LIN {X 0,Y 466.685,Z 325.228,A -85,B 0,C 180,E1 -7652.59,E2 -7652.59} C_VEL
LIN {X 0,Y 466.715,Z 322.29,A -85,B 0,C 180,E1 -7653.886,E2 -7653.886} C_VEL
LIN {X 0,Y 466.717,Z 319.594,A -85,B 0,C 180,E1 -7654.751,E2 -7654.751} C_VEL
LIN {X 0,Y 466.821,Z 316.273,A -85,B 0,C 180,E1 -7655.616,E2 -7655.616} C_VEL
LIN {X 0,Y 466.891,Z 311.9,A -85,B 0,C 180,E1 -7656.544,E2 -7656.544} C_VEL
LIN {X 0,Y 467.057,Z 305.94,A -85,B 0,C 180,E1 -7657.566,E2 -7657.566} C_VEL
LIN {X 0,Y 467.255,Z 299.775,A -85,B 0,C 180,E1 -7658.433,E2 -7658.433} C_VEL
LIN {X 0,Y 467.469,Z 293.294,A -85,B 0,C 180,E1 -7659.192,E2 -7659.192} C_VEL
LIN {X 0,Y 467.75,Z 285.446,A -85,B 0,C 180,E1 -7659.95,E2 -7659.95} C_VEL
LIN {X 0,Y 468.086,Z 277.17,A -85,B 0,C 180,E1 -7660.599,E2 -7660.599} C_VEL
LIN {X 0,Y 468.393,Z 266.639,A -85,B 0,C 180,E1 -7661.248,E2 -7661.248} C_VEL
LIN {X 0,Y 468.216,Z 258.863,A -85,B 0,C 180,E1 -7661.613,E2 -7661.613} C_VEL
LIN {X 0,Y 466.947,Z 246.747,A -85,B 0,C 180,E1 -7662.034,E2 -7662.034} C_VEL
LIN {X 0,Y 466.898,Z 245.995,A -85,B 0,C 180,E1 -7662.074,E2 -7662.074} C_VEL
LIN {X 0,Y 467.105,Z 234.959,A -85,B 0,C 180,E1 -7665.714,E2 -7665.714} C_VEL
LIN {X 0,Y 467.312,Z 226.159,A -85,B 0,C 180,E1 -7668.653,E2 -7668.653} C_VEL
LIN {X 0,Y 467.611,Z 217.438,A -85,B 0,C 180,E1 -7671.619,E2 -7671.619} C_VEL
LIN {X 0,Y 468.104,Z 206.857,A -85,B 0,C 180,E1 -7675.304,E2 -7675.304} C_VEL
LIN {X 0,Y 468.59,Z 197.452,A -85,B 0,C 180,E1 -7678.682,E2 -7678.682} C_VEL
LIN {X 0,Y 468.856,Z 190.408,A -85,B 0,C 180,E1 -7681.305,E2 -7681.305} C_VEL
LIN {X 0,Y 467.631,Z 183.051,A -85,B 0,C 180,E1 -7684.249,E2 -7684.249} C_VEL
LIN {X 0,Y 467.551,Z 183.059,A -85,B 0,C 180,E1 -7687.186,E2 -7687.186} C_VEL
LIN {X 0,Y 467.578,Z 183.056,A -85,B 0,C 180,E1 -7690.265,E2 -7690.265} C_VEL
LIN {X 0,Y 467.59,Z 183.054,A -85,B 0,C 180,E1 -7692.567,E2 -7692.567} C_VEL
LIN {X 0,Y 467.569,Z 183.056,A -85,B 0,C 180,E1 -7695.052,E2 -7695.052} C_VEL
LIN {X 0,Y 467.577,Z 183.055,A -85,B 0,C 180,E1 -7698.597,E2 -7698.597} C_VEL
LIN {X 0,Y 467.569,Z 183.058,A -85,B 0,C 180,E1 -7701.955,E2 -7701.955} C_VEL
LIN {X 0,Y 467.568,Z 183.054,A -85,B 0,C 180,E1 -7705.167,E2 -7705.167} C_VEL
LIN {X 0,Y 467.587,Z 183.056,A -85,B 0,C 180,E1 -7708.26,E2 -7708.26} C_VEL
LIN {X 0,Y 467.579,Z 183.055,A -85,B 0,C 180,E1 -7711.25,E2 -7711.25} C_VEL
LIN {X 0,Y 467.602,Z 183.053,A -85,B 0,C 180,E1 -7714.159,E2 -7714.159} C_VEL
LIN {X 0,Y 467.581,Z 183.054,A -85,B 0,C 180,E1 -7716.996,E2 -7716.996} C_VEL
LIN {X 0,Y 467.627,Z 183.051,A -85,B 0,C 180,E1 -7719.777,E2 -7719.777} C_VEL
LIN {X 0,Y 467.603,Z 183.051,A -85,B 0,C 180,E1 -7722.506,E2 -7722.506} C_VEL
LIN {X 0,Y 467.611,Z 183.052,A -85,B 0,C 180,E1 -7725.196,E2 -7725.196} C_VEL
LIN {X 0,Y 467.661,Z 183.045,A -85,B 0,C 180,E1 -7727.854,E2 -7727.854} C_VEL
LIN {X 0,Y 467.673,Z 183.045,A -85,B 0,C 180,E1 -7731.356,E2 -7731.356} C_VEL
LIN {X 0,Y 467.736,Z 183.035,A -85,B 0,C 180,E1 -7733.962,E2 -7733.962} C_VEL
LIN {X 0,Y 467.861,Z 183.022,A -85,B 0,C 180,E1 -7737.416,E2 -7737.416} C_VEL
LIN {X 0,Y 467.885,Z 183.017,A -85,B 0,C 180,E1 -7739.999,E2 -7739.999} C_VEL
LIN {X 0,Y 467.861,Z 183.019,A -85,B 0,C 180,E1 -7742.582,E2 -7742.582} C_VEL
LIN {X 0,Y 467.736,Z 183.033,A -85,B 0,C 180,E1 -7746.037,E2 -7746.037} C_VEL
LIN {X 0,Y 467.672,Z 183.043,A -85,B 0,C 180,E1 -7748.642,E2 -7748.642} C_VEL
LIN {X 0,Y 467.658,Z 183.045,A -85,B 0,C 180,E1 -7752.144,E2 -7752.144} C_VEL
LIN {X 0,Y 467.64,Z 183.047,A -85,B 0,C 180,E1 -7755.694,E2 -7755.694} C_VEL
LIN {X 0,Y 467.623,Z 183.05,A -85,B 0,C 180,E1 -7759.307,E2 -7759.307} C_VEL
LIN {X 0,Y 467.535,Z 183.062,A -85,B 0,C 180,E1 -7762.073,E2 -7762.073} C_VEL
LIN {X 0,Y 467.585,Z 183.054,A -85,B 0,C 180,E1 -7764.887,E2 -7764.887} C_VEL
LIN {X 0,Y 467.627,Z 183.048,A -85,B 0,C 180,E1 -7767.767,E2 -7767.767} C_VEL
LIN {X 0,Y 467.567,Z 183.056,A -85,B 0,C 180,E1 -7771.044,E2 -7771.044} C_VEL
LIN {X 0,Y 467.588,Z 183.054,A -85,B 0,C 180,E1 -7774.241,E2 -7774.241} C_VEL
LIN {X 0,Y 467.547,Z 183.059,A -85,B 0,C 180,E1 -7777.186,E2 -7777.186} C_VEL
LIN {X 0,Y 467.574,Z 183.056,A -85,B 0,C 180,E1 -7780.264,E2 -7780.264} C_VEL
LIN {X 0,Y 467.582,Z 183.054,A -85,B 0,C 180,E1 -7782.566,E2 -7782.566} C_VEL
LIN {X 0,Y 467.566,Z 183.056,A -85,B 0,C 180,E1 -7785.052,E2 -7785.052} C_VEL
LIN {X 0,Y 467.584,Z 183.055,A -85,B 0,C 180,E1 -7787.439,E2 -7787.439} C_VEL
LIN {X 0,Y 467.576,Z 183.054,A -85,B 0,C 180,E1 -7790.854,E2 -7790.854} C_VEL
LIN {X 0,Y 467.557,Z 183.057,A -85,B 0,C 180,E1 -7794.259,E2 -7794.259} C_VEL
LIN {X 0,Y 467.576,Z 183.055,A -85,B 0,C 180,E1 -7797.32,E2 -7797.32} C_VEL
LIN {X 0,Y 467.572,Z 183.055,A -85,B 0,C 180,E1 -7800.665,E2 -7800.665} C_VEL
LIN {X 0,Y 467.609,Z 183.052,A -85,B 0,C 180,E1 -7803.199,E2 -7803.199} C_VEL
LIN {X 0,Y 467.585,Z 183.054,A -85,B 0,C 180,E1 -7806.467,E2 -7806.467} C_VEL
LIN {X 0,Y 467.616,Z 183.05,A -85,B 0,C 180,E1 -7809.777,E2 -7809.777} C_VEL
LIN {X 0,Y 467.601,Z 183.051,A -85,B 0,C 180,E1 -7812.506,E2 -7812.506} C_VEL
LIN {X 0,Y 467.594,Z 183.052,A -85,B 0,C 180,E1 -7815.417,E2 -7815.417} C_VEL
LIN {X 0,Y 466.928,Z 183.134,A -85,B 0,C 180,E1 -7816.137,E2 -7816.137} C_VEL
LIN {X 0,Y 464.094,Z 183.489,A -85,B 0,C 180,E1 -7817.306,E2 -7817.306} C_VEL
LIN {X 0,Y 461.696,Z 183.788,A -85,B 0,C 180,E1 -7818.248,E2 -7818.248} C_VEL
LIN {X 0,Y 460.666,Z 183.917,A -85,B 0,C 180,E1 -7818.976,E2 -7818.976} C_VEL
LIN {X 0,Y 460.581,Z 183.926,A -85,B 0,C 180,E1 -7819.223,E2 -7819.223} C_VEL
LIN {X 0,Y 460.711,Z 183.91,A -85,B 0,C 180,E1 -7822.538,E2 -7822.538} C_VEL
LIN {X 0,Y 460.689,Z 183.915,A -85,B 0,C 180,E1 -7824.748,E2 -7824.748} C_VEL
LIN {X 0,Y 460.79,Z 183.9,A -85,B 0,C 180,E1 -7827.377,E2 -7827.377} C_VEL
LIN {X 0,Y 460.842,Z 183.894,A -85,B 0,C 180,E1 -7830,E2 -7830} C_VEL
LIN {X 0,Y 460.817,Z 183.898,A -85,B 0,C 180,E1 -7832.622,E2 -7832.622} C_VEL
LIN {X 0,Y 460.702,Z 183.913,A -85,B 0,C 180,E1 -7836.13,E2 -7836.13} C_VEL
LIN {X 0,Y 460.62,Z 183.922,A -85,B 0,C 180,E1 -7838.776,E2 -7838.776} C_VEL
LIN {X 0,Y 460.59,Z 183.928,A -85,B 0,C 180,E1 -7842.335,E2 -7842.335} C_VEL
LIN {X 0,Y 460.291,Z 184.096,A -85,B 0,C 180,E1 -7844.931,E2 -7844.931} C_VEL
LIN {X 0,Y 460.115,Z 188.342,A -85,B 0,C 180,E1 -7847.787,E2 -7847.787} C_VEL
LIN {X 0,Y 460.039,Z 192.537,A -85,B 0,C 180,E1 -7850.571,E2 -7850.571} C_VEL
LIN {X 0,Y 459.941,Z 197.069,A -85,B 0,C 180,E1 -7853.539,E2 -7853.539} C_VEL
LIN {X 0,Y 459.84,Z 201.353,A -85,B 0,C 180,E1 -7856.31,E2 -7856.31} C_VEL
LIN {X 0,Y 459.729,Z 206.164,A -85,B 0,C 180,E1 -7859.384,E2 -7859.384} C_VEL
LIN {X 0,Y 459.676,Z 211.565,A -85,B 0,C 180,E1 -7862.767,E2 -7862.767} C_VEL
LIN {X 0,Y 459.686,Z 213.246,A -85,B 0,C 180,E1 -7863.722,E2 -7863.722} C_VEL
LIN {X 0,Y 461.221,Z 222.711,A -85,B 0,C 180,E1 -7864.121,E2 -7864.121} C_VEL
LIN {X 0,Y 461.594,Z 228.119,A -85,B 0,C 180,E1 -7864.388,E2 -7864.388} C_VEL
LIN {X 0,Y 461.262,Z 237.826,A -85,B 0,C 180,E1 -7864.994,E2 -7864.994} C_VEL
LIN {X 0,Y 461.001,Z 245.945,A -85,B 0,C 180,E1 -7865.644,E2 -7865.644} C_VEL
LIN {X 0,Y 460.712,Z 254.566,A -85,B 0,C 180,E1 -7866.508,E2 -7866.508} C_VEL
LIN {X 0,Y 460.38,Z 262.083,A -85,B 0,C 180,E1 -7867.459,E2 -7867.459} C_VEL
LIN {X 0,Y 460.171,Z 268.447,A -85,B 0,C 180,E1 -7868.488,E2 -7868.488} C_VEL
LIN {X 0,Y 459.974,Z 272.818,A -85,B 0,C 180,E1 -7869.351,E2 -7869.351} C_VEL
LIN {X 0,Y 459.837,Z 276.248,A -85,B 0,C 180,E1 -7870.167,E2 -7870.167} C_VEL
LIN {X 0,Y 459.689,Z 280.407,A -85,B 0,C 180,E1 -7871.486,E2 -7871.486} C_VEL
LIN {X 0,Y 459.591,Z 283.196,A -85,B 0,C 180,E1 -7872.778,E2 -7872.778} C_VEL
LIN {X 0,Y 459.544,Z 284.733,A -85,B 0,C 180,E1 -7874.047,E2 -7874.047} C_VEL
LIN {X 0,Y 459.523,Z 285.066,A -85,B 0,C 180,E1 -7875.291,E2 -7875.291} C_VEL
LIN {X 0,Y 459.57,Z 284.346,A -85,B 0,C 180,E1 -7876.517,E2 -7876.517} C_VEL
LIN {X 0,Y 459.622,Z 282.626,A -85,B 0,C 180,E1 -7877.718,E2 -7877.718} C_VEL
LIN {X 0,Y 459.713,Z 279.899,A -85,B 0,C 180,E1 -7878.902,E2 -7878.902} C_VEL
LIN {X 0,Y 459.936,Z 274.892,A -85,B 0,C 180,E1 -7880.362,E2 -7880.362} C_VEL
LIN {X 0,Y 460.183,Z 269.452,A -85,B 0,C 180,E1 -7881.514,E2 -7881.514} C_VEL
LIN {X 0,Y 460.417,Z 263.346,A -85,B 0,C 180,E1 -7882.537,E2 -7882.537} C_VEL
LIN {X 0,Y 460.766,Z 255.068,A -85,B 0,C 180,E1 -7883.622,E2 -7883.622} C_VEL
LIN {X 0,Y 461.056,Z 246.575,A -85,B 0,C 180,E1 -7884.484,E2 -7884.484} C_VEL
LIN {X 0,Y 461.339,Z 238.745,A -85,B 0,C 180,E1 -7885.121,E2 -7885.121} C_VEL
LIN {X 0,Y 461.681,Z 229.369,A -85,B 0,C 180,E1 -7885.721,E2 -7885.721} C_VEL
LIN {X 0,Y 461.438,Z 223.284,A -85,B 0,C 180,E1 -7886.03,E2 -7886.03} C_VEL
LIN {X 0,Y 459.731,Z 213.544,A -85,B 0,C 180,E1 -7886.48,E2 -7886.48} C_VEL
LIN {X 0,Y 459.77,Z 208.543,A -85,B 0,C 180,E1 -7889.707,E2 -7889.707} C_VEL
LIN {X 0,Y 459.922,Z 203.907,A -85,B 0,C 180,E1 -7892.716,E2 -7892.716} C_VEL
LIN {X 0,Y 460,Z 199.515,A -85,B 0,C 180,E1 -7895.638,E2 -7895.638} C_VEL
LIN {X 0,Y 460.104,Z 194.897,A -85,B 0,C 180,E1 -7898.711,E2 -7898.711} C_VEL
LIN {X 0,Y 460.227,Z 191.101,A -85,B 0,C 180,E1 -7901.297,E2 -7901.297} C_VEL
LIN {X 0,Y 460.332,Z 186.977,A -85,B 0,C 180,E1 -7904.12,E2 -7904.12} C_VEL
LIN {X 0,Y 460.347,Z 184.5,A -85,B 0,C 180,E1 -7905.862,E2 -7905.862} C_VEL
LIN {X 0,Y 460.432,Z 183.952,A -85,B 0,C 180,E1 -7906.765,E2 -7906.765} C_VEL
LIN {X 0,Y 460.603,Z 183.928,A -85,B 0,C 180,E1 -7908.56,E2 -7908.56} C_VEL
LIN {X 0,Y 460.696,Z 183.917,A -85,B 0,C 180,E1 -7912.109,E2 -7912.109} C_VEL
LIN {X 0,Y 460.697,Z 183.917,A -85,B 0,C 180,E1 -7914.749,E2 -7914.749} C_VEL
LIN {X 0,Y 460.801,Z 183.901,A -85,B 0,C 180,E1 -7917.378,E2 -7917.378} C_VEL
LIN {X 0,Y 460.855,Z 183.894,A -85,B 0,C 180,E1 -7920.001,E2 -7920.001} C_VEL
LIN {X 0,Y 460.801,Z 183.9,A -85,B 0,C 180,E1 -7922.623,E2 -7922.623} C_VEL
LIN {X 0,Y 460.709,Z 183.912,A -85,B 0,C 180,E1 -7926.131,E2 -7926.131} C_VEL
LIN {X 0,Y 460.622,Z 183.921,A -85,B 0,C 180,E1 -7928.777,E2 -7928.777} C_VEL
LIN {X 0,Y 460.616,Z 183.923,A -85,B 0,C 180,E1 -7932.445,E2 -7932.445} C_VEL
LIN {X 0,Y 460.603,Z 183.925,A -85,B 0,C 180,E1 -7935.998,E2 -7935.998} C_VEL
LIN {X 0,Y 460.574,Z 183.927,A -85,B 0,C 180,E1 -7938.902,E2 -7938.902} C_VEL
LIN {X 0,Y 460.518,Z 183.935,A -85,B 0,C 180,E1 -7941.486,E2 -7941.486} C_VEL
LIN {X 0,Y 460.533,Z 183.934,A -85,B 0,C 180,E1 -7944.333,E2 -7944.333} C_VEL
LIN {X 0,Y 460.574,Z 183.928,A -85,B 0,C 180,E1 -7947.244,E2 -7947.244} C_VEL
LIN {X 0,Y 460.513,Z 183.936,A -85,B 0,C 180,E1 -7950.24,E2 -7950.24} C_VEL
LIN {X 0,Y 460.531,Z 183.934,A -85,B 0,C 180,E1 -7953.325,E2 -7953.325} C_VEL
LIN {X 0,Y 460.478,Z 183.939,A -85,B 0,C 180,E1 -7956.53,E2 -7956.53} C_VEL
LIN {X 0,Y 460.529,Z 183.934,A -85,B 0,C 180,E1 -7959.863,E2 -7959.863} C_VEL
LIN {X 0,Y 460.515,Z 183.938,A -85,B 0,C 180,E1 -7962.901,E2 -7962.901} C_VEL
LIN {X 0,Y 460.513,Z 183.938,A -85,B 0,C 180,E1 -7965.831,E2 -7965.831} C_VEL
LIN {X 0,Y 460.533,Z 183.934,A -85,B 0,C 180,E1 -7968.989,E2 -7968.989} C_VEL
LIN {X 0,Y 460.528,Z 183.934,A -85,B 0,C 180,E1 -7971.267,E2 -7971.267} C_VEL
LIN {X 0,Y 460.597,Z 184.056,A -85,B 0,C 180,E1 -7975.122,E2 -7975.122} C_VEL
LIN {X 0,Y 461.662,Z 190.143,A -85,B 0,C 180,E1 -7977.804,E2 -7977.804} C_VEL
LIN {X 0,Y 461.924,Z 193.849,A -85,B 0,C 180,E1 -7979.357,E2 -7979.357} C_VEL
LIN {X 0,Y 461.46,Z 200.744,A -85,B 0,C 180,E1 -7982.048,E2 -7982.048} C_VEL
LIN {X 0,Y 460.944,Z 209.202,A -85,B 0,C 180,E1 -7985.21,E2 -7985.21} C_VEL
LIN {X 0,Y 460.517,Z 218.574,A -85,B 0,C 180,E1 -7988.58,E2 -7988.58} C_VEL
LIN {X 0,Y 460.219,Z 227.7,A -85,B 0,C 180,E1 -7991.757,E2 -7991.757} C_VEL
LIN {X 0,Y 459.936,Z 237.099,A -85,B 0,C 180,E1 -7994.944,E2 -7994.944} C_VEL
LIN {X 0,Y 459.794,Z 245.407,A -85,B 0,C 180,E1 -7997.718,E2 -7997.718} C_VEL
LIN {X 0,Y 461.037,Z 256.939,A -85,B 0,C 180,E1 -7998.115,E2 -7998.115} C_VEL
LIN {X 0,Y 461.463,Z 265.358,A -85,B 0,C 180,E1 -7998.514,E2 -7998.514} C_VEL
LIN {X 0,Y 461.153,Z 275.468,A -85,B 0,C 180,E1 -7999.129,E2 -7999.129} C_VEL
LIN {X 0,Y 460.817,Z 283.943,A -85,B 0,C 180,E1 -7999.788,E2 -7999.788} C_VEL
LIN {X 0,Y 460.479,Z 291.949,A -85,B 0,C 180,E1 -8000.557,E2 -8000.557} C_VEL
LIN {X 0,Y 460.283,Z 297.713,A -85,B 0,C 180,E1 -8001.217,E2 -8001.217} C_VEL
LIN {X 0,Y 460.046,Z 304.151,A -85,B 0,C 180,E1 -8002.097,E2 -8002.097} C_VEL
LIN {X 0,Y 459.874,Z 309.506,A -85,B 0,C 180,E1 -8002.978,E2 -8002.978} C_VEL
LIN {X 0,Y 459.727,Z 313.972,A -85,B 0,C 180,E1 -8003.857,E2 -8003.857} C_VEL
LIN {X 0,Y 459.648,Z 319.232,A -85,B 0,C 180,E1 -8005.176,E2 -8005.176} C_VEL
LIN {X 0,Y 459.608,Z 321.926,A -85,B 0,C 180,E1 -8006.054,E2 -8006.054} C_VEL
LIN {X 0,Y 459.608,Z 324.883,A -85,B 0,C 180,E1 -8007.371,E2 -8007.371} C_VEL
LIN {X 0,Y 459.57,Z 326.159,A -85,B 0,C 180,E1 -8008.247,E2 -8008.247} C_VEL
LIN {X 0,Y 459.555,Z 326.952,A -85,B 0,C 180,E1 -8009.124,E2 -8009.124} C_VEL
LIN {X 0,Y 459.536,Z 327.255,A -85,B 0,C 180,E1 -8010,E2 -8010} C_VEL
LIN {X 0,Y 459.554,Z 326.966,A -85,B 0,C 180,E1 -8010.876,E2 -8010.876} C_VEL
LIN {X 0,Y 459.57,Z 326.17,A -85,B 0,C 180,E1 -8011.753,E2 -8011.753} C_VEL
LIN {X 0,Y 459.608,Z 324.891,A -85,B 0,C 180,E1 -8012.629,E2 -8012.629} C_VEL
LIN {X 0,Y 459.608,Z 321.944,A -85,B 0,C 180,E1 -8013.946,E2 -8013.946} C_VEL
LIN {X 0,Y 459.708,Z 317.717,A -85,B 0,C 180,E1 -8015.263,E2 -8015.263} C_VEL
LIN {X 0,Y 459.787,Z 312.24,A -85,B 0,C 180,E1 -8016.511,E2 -8016.511} C_VEL
LIN {X 0,Y 459.973,Z 306.973,A -85,B 0,C 180,E1 -8017.462,E2 -8017.462} C_VEL
LIN {X 0,Y 460.158,Z 301.075,A -85,B 0,C 180,E1 -8018.343,E2 -8018.343} C_VEL
LIN {X 0,Y 460.394,Z 293.889,A -85,B 0,C 180,E1 -8019.224,E2 -8019.224} C_VEL
LIN {X 0,Y 460.69,Z 286.224,A -85,B 0,C 180,E1 -8019.993,E2 -8019.993} C_VEL
LIN {X 0,Y 461.017,Z 278.183,A -85,B 0,C 180,E1 -8020.652,E2 -8020.652} C_VEL
LIN {X 0,Y 461.308,Z 269.861,A -85,B 0,C 180,E1 -8021.201,E2 -8021.201} C_VEL
LIN {X 0,Y 461.393,Z 261.973,A -85,B 0,C 180,E1 -8021.616,E2 -8021.616} C_VEL
LIN {X 0,Y 460.567,Z 252.737,A -85,B 0,C 180,E1 -8022.005,E2 -8022.005} C_VEL
LIN {X 0,Y 459.819,Z 245.782,A -85,B 0,C 180,E1 -8022.243,E2 -8022.243} C_VEL
LIN {X 0,Y 460.019,Z 235.34,A -85,B 0,C 180,E1 -8025.742,E2 -8025.742} C_VEL
LIN {X 0,Y 460.301,Z 225.435,A -85,B 0,C 180,E1 -8029.118,E2 -8029.118} C_VEL
LIN {X 0,Y 460.666,Z 215.947,A -85,B 0,C 180,E1 -8032.421,E2 -8032.421} C_VEL
LIN {X 0,Y 461.142,Z 206.045,A -85,B 0,C 180,E1 -8035.948,E2 -8035.948} C_VEL
LIN {X 0,Y 461.641,Z 197.323,A -85,B 0,C 180,E1 -8039.155,E2 -8039.155} C_VEL
LIN {X 0,Y 461.855,Z 192.028,A -85,B 0,C 180,E1 -8041.157,E2 -8041.157} C_VEL
LIN {X 0,Y 460.822,Z 185.428,A -85,B 0,C 180,E1 -8043.826,E2 -8043.826} C_VEL
LIN {X 0,Y 460.564,Z 183.93,A -85,B 0,C 180,E1 -8044.511,E2 -8044.511} C_VEL
LIN {X 0,Y 460.504,Z 183.938,A -85,B 0,C 180,E1 -8047.623,E2 -8047.623} C_VEL
LIN {X 0,Y 460.542,Z 183.932,A -85,B 0,C 180,E1 -8050.269,E2 -8050.269} C_VEL
LIN {X 0,Y 460.502,Z 183.935,A -85,B 0,C 180,E1 -8053.376,E2 -8053.376} C_VEL
LIN {X 0,Y 460.512,Z 183.938,A -85,B 0,C 180,E1 -8056.626,E2 -8056.626} C_VEL
LIN {X 0,Y 460.538,Z 183.933,A -85,B 0,C 180,E1 -8059.732,E2 -8059.732} C_VEL
LIN {X 0,Y 460.503,Z 183.936,A -85,B 0,C 180,E1 -8062.524,E2 -8062.524} C_VEL
LIN {X 0,Y 460.551,Z 183.93,A -85,B 0,C 180,E1 -8065.624,E2 -8065.624} C_VEL
LIN {X 0,Y 460.542,Z 183.93,A -85,B 0,C 180,E1 -8068.744,E2 -8068.744} C_VEL
LIN {X 0,Y 460.585,Z 183.927,A -85,B 0,C 180,E1 -8072.254,E2 -8072.254} C_VEL
LIN {X 0,Y 460.544,Z 183.931,A -85,B 0,C 180,E1 -8074.704,E2 -8074.704} C_VEL
LIN {X 0,Y 460.515,Z 183.936,A -85,B 0,C 180,E1 -8077.571,E2 -8077.571} C_VEL
LIN {X 0,Y 460.573,Z 183.927,A -85,B 0,C 180,E1 -8080.384,E2 -8080.384} C_VEL
LIN {X 0,Y 460.605,Z 183.923,A -85,B 0,C 180,E1 -8084.002,E2 -8084.002} C_VEL
LIN {X 0,Y 460.614,Z 183.923,A -85,B 0,C 180,E1 -8087.665,E2 -8087.665} C_VEL
LIN {X 0,Y 460.623,Z 183.923,A -85,B 0,C 180,E1 -8091.223,E2 -8091.223} C_VEL
LIN {X 0,Y 460.702,Z 183.912,A -85,B 0,C 180,E1 -8093.869,E2 -8093.869} C_VEL
LIN {X 0,Y 460.802,Z 183.901,A -85,B 0,C 180,E1 -8097.377,E2 -8097.377} C_VEL
LIN {X 0,Y 460.855,Z 183.892,A -85,B 0,C 180,E1 -8099.999,E2 -8099.999} C_VEL
LIN {X 0,Y 460.802,Z 183.899,A -85,B 0,C 180,E1 -8102.622,E2 -8102.622} C_VEL
LIN {X 0,Y 460.702,Z 183.91,A -85,B 0,C 180,E1 -8106.129,E2 -8106.129} C_VEL
LIN {X 0,Y 460.622,Z 183.922,A -85,B 0,C 180,E1 -8108.775,E2 -8108.775} C_VEL
LIN {X 0,Y 460.616,Z 183.922,A -85,B 0,C 180,E1 -8112.444,E2 -8112.444} C_VEL
LIN {X 0,Y 460.602,Z 183.924,A -85,B 0,C 180,E1 -8115.997,E2 -8115.997} C_VEL
LIN {X 0,Y 460.569,Z 183.927,A -85,B 0,C 180,E1 -8119.614,E2 -8119.614} C_VEL
LIN {X 0,Y 460.511,Z 183.936,A -85,B 0,C 180,E1 -8122.428,E2 -8122.428} C_VEL
LIN {X 0,Y 460.552,Z 183.93,A -85,B 0,C 180,E1 -8125.797,E2 -8125.797} C_VEL
LIN {X 0,Y 460.555,Z 183.931,A -85,B 0,C 180,E1 -8128.232,E2 -8128.232} C_VEL
LIN {X 0,Y 460.52,Z 183.933,A -85,B 0,C 180,E1 -8131.282,E2 -8131.282} C_VEL
LIN {X 0,Y 460.532,Z 183.935,A -85,B 0,C 180,E1 -8134.505,E2 -8134.505} C_VEL
LIN {X 0,Y 460.525,Z 183.934,A -85,B 0,C 180,E1 -8137.619,E2 -8137.619} C_VEL
LIN {X 0,Y 460.538,Z 183.932,A -85,B 0,C 180,E1 -8140.268,E2 -8140.268} C_VEL
LIN {X 0,Y 460.495,Z 183.936,A -85,B 0,C 180,E1 -8143.374,E2 -8143.374} C_VEL
LIN {X 0,Y 460.495,Z 183.936,A -85,B 0,C 180,E1 -8146.624,E2 -8146.624} C_VEL
LIN {X 0,Y 460.536,Z 183.933,A -85,B 0,C 180,E1 -8149.73,E2 -8149.73} C_VEL
LIN {X 0,Y 460.521,Z 183.934,A -85,B 0,C 180,E1 -8152.518,E2 -8152.518} C_VEL
LIN {X 0,Y 460.543,Z 183.932,A -85,B 0,C 180,E1 -8155.623,E2 -8155.623} C_VEL
LIN {X 0,Y 460.53,Z 183.932,A -85,B 0,C 180,E1 -8158.744,E2 -8158.744} C_VEL
LIN {X 0,Y 460.551,Z 183.931,A -85,B 0,C 180,E1 -8161.767,E2 -8161.767} C_VEL
LIN {X 0,Y 460.551,Z 183.929,A -85,B 0,C 180,E1 -8164.705,E2 -8164.705} C_VEL
LIN {X 0,Y 460.505,Z 183.938,A -85,B 0,C 180,E1 -8167.571,E2 -8167.571} C_VEL
LIN {X 0,Y 460.562,Z 183.929,A -85,B 0,C 180,E1 -8170.384,E2 -8170.384} C_VEL
LIN {X 0,Y 460.557,Z 183.931,A -85,B 0,C 180,E1 -8173.146,E2 -8173.146} C_VEL
LIN {X 0,Y 460.554,Z 183.928,A -85,B 0,C 180,E1 -8175.868,E2 -8175.868} C_VEL
LIN {X 0,Y 460.625,Z 183.922,A -85,B 0,C 180,E1 -8178.559,E2 -8178.559} C_VEL
LIN {X 0,Y 460.581,Z 183.926,A -85,B 0,C 180,E1 -8179.223,E2 -8179.223} C_VEL
LIN {X 0,Y 459.917,Z 184.011,A -85,B 0,C 180,E1 -8179.953,E2 -8179.953} C_VEL
LIN {X 0,Y 457.095,Z 184.366,A -85,B 0,C 180,E1 -8181.139,E2 -8181.139} C_VEL
LIN {X 0,Y 454.716,Z 184.661,A -85,B 0,C 180,E1 -8182.096,E2 -8182.096} C_VEL
LIN {X 0,Y 453.705,Z 184.784,A -85,B 0,C 180,E1 -8182.835,E2 -8182.835} C_VEL
LIN {X 0,Y 453.628,Z 184.792,A -85,B 0,C 180,E1 -8183.085,E2 -8183.085} C_VEL
LIN {X 0,Y 453.663,Z 184.79,A -85,B 0,C 180,E1 -8184.666,E2 -8184.666} C_VEL
LIN {X 0,Y 453.735,Z 184.779,A -85,B 0,C 180,E1 -8187.336,E2 -8187.336} C_VEL
LIN {X 0,Y 453.813,Z 184.77,A -85,B 0,C 180,E1 -8190,E2 -8190} C_VEL
LIN {X 0,Y 453.757,Z 184.777,A -85,B 0,C 180,E1 -8192.663,E2 -8192.663} C_VEL
LIN {X 0,Y 453.669,Z 184.789,A -85,B 0,C 180,E1 -8196.225,E2 -8196.225} C_VEL
LIN {X 0,Y 453.584,Z 184.798,A -85,B 0,C 180,E1 -8198.913,E2 -8198.913} C_VEL
LIN {X 0,Y 453.52,Z 184.807,A -85,B 0,C 180,E1 -8202.51,E2 -8202.51} C_VEL
LIN {X 0,Y 453.24,Z 184.917,A -85,B 0,C 180,E1 -8204.939,E2 -8204.939} C_VEL
LIN {X 0,Y 453.064,Z 189.527,A -85,B 0,C 180,E1 -8208.074,E2 -8208.074} C_VEL
LIN {X 0,Y 452.965,Z 194.538,A -85,B 0,C 180,E1 -8211.423,E2 -8211.423} C_VEL
LIN {X 0,Y 452.858,Z 199.622,A -85,B 0,C 180,E1 -8214.773,E2 -8214.773} C_VEL
LIN {X 0,Y 452.72,Z 204.247,A -85,B 0,C 180,E1 -8217.768,E2 -8217.768} C_VEL
LIN {X 0,Y 452.599,Z 209.03,A -85,B 0,C 180,E1 -8220.826,E2 -8220.826} C_VEL
LIN {X 0,Y 452.595,Z 213.297,A -85,B 0,C 180,E1 -8223.539,E2 -8223.539} C_VEL
LIN {X 0,Y 454.246,Z 223.477,A -85,B 0,C 180,E1 -8223.981,E2 -8223.981} C_VEL
LIN {X 0,Y 454.638,Z 228.12,A -85,B 0,C 180,E1 -8224.215,E2 -8224.215} C_VEL
LIN {X 0,Y 454.281,Z 238.116,A -85,B 0,C 180,E1 -8224.846,E2 -8224.846} C_VEL
LIN {X 0,Y 454.016,Z 246.002,A -85,B 0,C 180,E1 -8225.485,E2 -8225.485} C_VEL
LIN {X 0,Y 453.764,Z 253.171,A -85,B 0,C 180,E1 -8226.199,E2 -8226.199} C_VEL
LIN {X 0,Y 453.392,Z 261.293,A -85,B 0,C 180,E1 -8227.195,E2 -8227.195} C_VEL
LIN {X 0,Y 453.117,Z 268.496,A -85,B 0,C 180,E1 -8228.346,E2 -8228.346} C_VEL
LIN {X 0,Y 452.857,Z 274.183,A -85,B 0,C 180,E1 -8229.516,E2 -8229.516} C_VEL
LIN {X 0,Y 452.682,Z 278.611,A -85,B 0,C 180,E1 -8230.697,E2 -8230.697} C_VEL
LIN {X 0,Y 452.577,Z 281.894,A -85,B 0,C 180,E1 -8231.893,E2 -8231.893} C_VEL
LIN {X 0,Y 452.494,Z 284.071,A -85,B 0,C 180,E1 -8233.116,E2 -8233.116} C_VEL
LIN {X 0,Y 452.434,Z 285.21,A -85,B 0,C 180,E1 -8234.395,E2 -8234.395} C_VEL
LIN {X 0,Y 452.434,Z 285.277,A -85,B 0,C 180,E1 -8235.653,E2 -8235.653} C_VEL
LIN {X 0,Y 452.497,Z 284.312,A -85,B 0,C 180,E1 -8236.892,E2 -8236.892} C_VEL
LIN {X 0,Y 452.584,Z 282.186,A -85,B 0,C 180,E1 -8238.191,E2 -8238.191} C_VEL
LIN {X 0,Y 452.716,Z 278.58,A -85,B 0,C 180,E1 -8239.524,E2 -8239.524} C_VEL
LIN {X 0,Y 452.962,Z 273.436,A -85,B 0,C 180,E1 -8240.876,E2 -8240.876} C_VEL
LIN {X 0,Y 453.219,Z 267.857,A -85,B 0,C 180,E1 -8241.994,E2 -8241.994} C_VEL
LIN {X 0,Y 453.512,Z 261.108,A -85,B 0,C 180,E1 -8243.04,E2 -8243.04} C_VEL
LIN {X 0,Y 453.825,Z 253.737,A -85,B 0,C 180,E1 -8243.953,E2 -8243.953} C_VEL
LIN {X 0,Y 454.121,Z 246.711,A -85,B 0,C 180,E1 -8244.663,E2 -8244.663} C_VEL
LIN {X 0,Y 454.403,Z 238.152,A -85,B 0,C 180,E1 -8245.363,E2 -8245.363} C_VEL
LIN {X 0,Y 454.796,Z 227.944,A -85,B 0,C 180,E1 -8246,E2 -8246} C_VEL
LIN {X 0,Y 453.875,Z 220.518,A -85,B 0,C 180,E1 -8246.381,E2 -8246.381} C_VEL
LIN {X 0,Y 452.66,Z 213.836,A -85,B 0,C 180,E1 -8246.678,E2 -8246.678} C_VEL
LIN {X 0,Y 452.708,Z 208.412,A -85,B 0,C 180,E1 -8250.214,E2 -8250.214} C_VEL
LIN {X 0,Y 452.829,Z 203.821,A -85,B 0,C 180,E1 -8253.252,E2 -8253.252} C_VEL
LIN {X 0,Y 452.951,Z 199.321,A -85,B 0,C 180,E1 -8256.269,E2 -8256.269} C_VEL
LIN {X 0,Y 453.055,Z 195.171,A -85,B 0,C 180,E1 -8259.098,E2 -8259.098} C_VEL
LIN {X 0,Y 453.182,Z 191.048,A -85,B 0,C 180,E1 -8261.932,E2 -8261.932} C_VEL
LIN {X 0,Y 453.327,Z 187.069,A -85,B 0,C 180,E1 -8264.72,E2 -8264.72} C_VEL
LIN {X 0,Y 453.358,Z 184.833,A -85,B 0,C 180,E1 -8266.555,E2 -8266.555} C_VEL
LIN {X 0,Y 453.552,Z 184.806,A -85,B 0,C 180,E1 -8268.38,E2 -8268.38} C_VEL
LIN {X 0,Y 453.653,Z 184.794,A -85,B 0,C 180,E1 -8271.986,E2 -8271.986} C_VEL
LIN {X 0,Y 453.671,Z 184.793,A -85,B 0,C 180,E1 -8274.668,E2 -8274.668} C_VEL
LIN {X 0,Y 453.745,Z 184.78,A -85,B 0,C 180,E1 -8277.337,E2 -8277.337} C_VEL
LIN {X 0,Y 453.825,Z 184.769,A -85,B 0,C 180,E1 -8280.001,E2 -8280.001} C_VEL
LIN {X 0,Y 453.745,Z 184.779,A -85,B 0,C 180,E1 -8282.664,E2 -8282.664} C_VEL
LIN {X 0,Y 453.675,Z 184.788,A -85,B 0,C 180,E1 -8286.226,E2 -8286.226} C_VEL
LIN {X 0,Y 453.588,Z 184.798,A -85,B 0,C 180,E1 -8288.914,E2 -8288.914} C_VEL
LIN {X 0,Y 453.566,Z 184.802,A -85,B 0,C 180,E1 -8292.529,E2 -8292.529} C_VEL
LIN {X 0,Y 453.547,Z 184.804,A -85,B 0,C 180,E1 -8296.196,E2 -8296.196} C_VEL
LIN {X 0,Y 453.523,Z 184.805,A -85,B 0,C 180,E1 -8299.041,E2 -8299.041} C_VEL
LIN {X 0,Y 453.479,Z 184.813,A -85,B 0,C 180,E1 -8301.837,E2 -8301.837} C_VEL
LIN {X 0,Y 453.503,Z 184.808,A -85,B 0,C 180,E1 -8304.736,E2 -8304.736} C_VEL
LIN {X 0,Y 453.535,Z 184.805,A -85,B 0,C 180,E1 -8307.96,E2 -8307.96} C_VEL
LIN {X 0,Y 453.468,Z 184.813,A -85,B 0,C 180,E1 -8311.526,E2 -8311.526} C_VEL
LIN {X 0,Y 453.49,Z 184.811,A -85,B 0,C 180,E1 -8314.778,E2 -8314.778} C_VEL
LIN {X 0,Y 453.465,Z 184.814,A -85,B 0,C 180,E1 -8318.312,E2 -8318.312} C_VEL
LIN {X 0,Y 453.496,Z 184.812,A -85,B 0,C 180,E1 -8320.609,E2 -8320.609} C_VEL
LIN {X 0,Y 453.458,Z 184.816,A -85,B 0,C 180,E1 -8323.244,E2 -8323.244} C_VEL
LIN {X 0,Y 453.468,Z 184.816,A -85,B 0,C 180,E1 -8325.779,E2 -8325.779} C_VEL
LIN {X 0,Y 453.481,Z 184.814,A -85,B 0,C 180,E1 -8328.21,E2 -8328.21} C_VEL
LIN {X 0,Y 453.512,Z 184.81,A -85,B 0,C 180,E1 -8330.791,E2 -8330.791} C_VEL
LIN {X 0,Y 453.496,Z 184.817,A -85,B 0,C 180,E1 -8334.468,E2 -8334.468} C_VEL
LIN {X 0,Y 453.566,Z 185.013,A -85,B 0,C 180,E1 -8334.883,E2 -8334.883} C_VEL
LIN {X 0,Y 454.68,Z 191.355,A -85,B 0,C 180,E1 -8337.768,E2 -8337.768} C_VEL
LIN {X 0,Y 454.937,Z 195.138,A -85,B 0,C 180,E1 -8339.35,E2 -8339.35} C_VEL
LIN {X 0,Y 454.364,Z 202.672,A -85,B 0,C 180,E1 -8342.352,E2 -8342.352} C_VEL
LIN {X 0,Y 453.826,Z 211.536,A -85,B 0,C 180,E1 -8345.713,E2 -8345.713} C_VEL
LIN {X 0,Y 453.414,Z 220.904,A -85,B 0,C 180,E1 -8349.114,E2 -8349.114} C_VEL
LIN {X 0,Y 453.117,Z 228.837,A -85,B 0,C 180,E1 -8351.928,E2 -8351.928} C_VEL
LIN {X 0,Y 452.849,Z 238.207,A -85,B 0,C 180,E1 -8355.163,E2 -8355.163} C_VEL
LIN {X 0,Y 452.723,Z 245.094,A -85,B 0,C 180,E1 -8357.505,E2 -8357.505} C_VEL
LIN {X 0,Y 454.109,Z 258.205,A -85,B 0,C 180,E1 -8357.996,E2 -8357.996} C_VEL
LIN {X 0,Y 454.453,Z 266.31,A -85,B 0,C 180,E1 -8358.402,E2 -8358.402} C_VEL
LIN {X 0,Y 454.1,Z 276.697,A -85,B 0,C 180,E1 -8359.071,E2 -8359.071} C_VEL
LIN {X 0,Y 453.799,Z 283.663,A -85,B 0,C 180,E1 -8359.628,E2 -8359.628} C_VEL
LIN {X 0,Y 453.476,Z 291.663,A -85,B 0,C 180,E1 -8360.41,E2 -8360.41} C_VEL
LIN {X 0,Y 453.254,Z 297.421,A -85,B 0,C 180,E1 -8361.08,E2 -8361.08} C_VEL
LIN {X 0,Y 452.988,Z 303.855,A -85,B 0,C 180,E1 -8361.974,E2 -8361.974} C_VEL
LIN {X 0,Y 452.802,Z 309.204,A -85,B 0,C 180,E1 -8362.867,E2 -8362.867} C_VEL
LIN {X 0,Y 452.652,Z 313.665,A -85,B 0,C 180,E1 -8363.761,E2 -8363.761} C_VEL
LIN {X 0,Y 452.579,Z 318.922,A -85,B 0,C 180,E1 -8365.101,E2 -8365.101} C_VEL
LIN {X 0,Y 452.506,Z 321.612,A -85,B 0,C 180,E1 -8365.992,E2 -8365.992} C_VEL
LIN {X 0,Y 452.533,Z 324.567,A -85,B 0,C 180,E1 -8367.33,E2 -8367.33} C_VEL
LIN {X 0,Y 452.483,Z 325.839,A -85,B 0,C 180,E1 -8368.22,E2 -8368.22} C_VEL
LIN {X 0,Y 452.489,Z 326.629,A -85,B 0,C 180,E1 -8369.11,E2 -8369.11} C_VEL
LIN {X 0,Y 452.469,Z 326.93,A -85,B 0,C 180,E1 -8370,E2 -8370} C_VEL
LIN {X 0,Y 452.489,Z 326.64,A -85,B 0,C 180,E1 -8370.89,E2 -8370.89} C_VEL
LIN {X 0,Y 452.483,Z 325.837,A -85,B 0,C 180,E1 -8371.78,E2 -8371.78} C_VEL
LIN {X 0,Y 452.533,Z 324.552,A -85,B 0,C 180,E1 -8372.671,E2 -8372.671} C_VEL
LIN {X 0,Y 452.506,Z 321.597,A -85,B 0,C 180,E1 -8374.008,E2 -8374.008} C_VEL
LIN {X 0,Y 452.62,Z 317.36,A -85,B 0,C 180,E1 -8375.346,E2 -8375.346} C_VEL
LIN {X 0,Y 452.731,Z 311.479,A -85,B 0,C 180,E1 -8376.686,E2 -8376.686} C_VEL
LIN {X 0,Y 452.89,Z 306.576,A -85,B 0,C 180,E1 -8377.58,E2 -8377.58} C_VEL
LIN {X 0,Y 453.096,Z 300.659,A -85,B 0,C 180,E1 -8378.474,E2 -8378.474} C_VEL
LIN {X 0,Y 453.358,Z 293.449,A -85,B 0,C 180,E1 -8379.368,E2 -8379.368} C_VEL
LIN {X 0,Y 453.685,Z 285.756,A -85,B 0,C 180,E1 -8380.149,E2 -8380.149} C_VEL
LIN {X 0,Y 454.034,Z 277.676,A -85,B 0,C 180,E1 -8380.818,E2 -8380.818} C_VEL
LIN {X 0,Y 454.324,Z 269.3,A -85,B 0,C 180,E1 -8381.375,E2 -8381.375} C_VEL
LIN {X 0,Y 454.352,Z 262.005,A -85,B 0,C 180,E1 -8381.767,E2 -8381.767} C_VEL
LIN {X 0,Y 453.525,Z 252.729,A -85,B 0,C 180,E1 -8382.167,E2 -8382.167} C_VEL
LIN {X 0,Y 452.711,Z 245.571,A -85,B 0,C 180,E1 -8382.401,E2 -8382.401} C_VEL
LIN {X 0,Y 452.948,Z 235.508,A -85,B 0,C 180,E1 -8385.845,E2 -8385.845} C_VEL
LIN {X 0,Y 453.28,Z 225.088,A -85,B 0,C 180,E1 -8389.473,E2 -8389.473} C_VEL
LIN {X 0,Y 453.657,Z 215.746,A -85,B 0,C 180,E1 -8392.787,E2 -8392.787} C_VEL
LIN {X 0,Y 454.138,Z 206.479,A -85,B 0,C 180,E1 -8396.158,E2 -8396.158} C_VEL
LIN {X 0,Y 454.683,Z 197.156,A -85,B 0,C 180,E1 -8399.645,E2 -8399.645} C_VEL
LIN {X 0,Y 454.859,Z 193.215,A -85,B 0,C 180,E1 -8401.172,E2 -8401.172} C_VEL
LIN {X 0,Y 453.839,Z 186.62,A -85,B 0,C 180,E1 -8403.882,E2 -8403.882} C_VEL
LIN {X 0,Y 453.514,Z 184.808,A -85,B 0,C 180,E1 -8404.701,E2 -8404.701} C_VEL
LIN {X 0,Y 453.466,Z 184.814,A -85,B 0,C 180,E1 -8408.312,E2 -8408.312} C_VEL
LIN {X 0,Y 453.497,Z 184.81,A -85,B 0,C 180,E1 -8410.609,E2 -8410.609} C_VEL
LIN {X 0,Y 453.458,Z 184.812,A -85,B 0,C 180,E1 -8413.244,E2 -8413.244} C_VEL
LIN {X 0,Y 453.464,Z 184.814,A -85,B 0,C 180,E1 -8415.778,E2 -8415.778} C_VEL
LIN {X 0,Y 453.497,Z 184.809,A -85,B 0,C 180,E1 -8419.409,E2 -8419.409} C_VEL
LIN {X 0,Y 453.456,Z 184.815,A -85,B 0,C 180,E1 -8422.81,E2 -8422.81} C_VEL
LIN {X 0,Y 453.481,Z 184.812,A -85,B 0,C 180,E1 -8426.087,E2 -8426.087} C_VEL
LIN {X 0,Y 453.481,Z 184.809,A -85,B 0,C 180,E1 -8429.24,E2 -8429.24} C_VEL
LIN {X 0,Y 453.54,Z 184.804,A -85,B 0,C 180,E1 -8432.297,E2 -8432.297} C_VEL
LIN {X 0,Y 453.505,Z 184.808,A -85,B 0,C 180,E1 -8435.265,E2 -8435.265} C_VEL
LIN {X 0,Y 453.485,Z 184.811,A -85,B 0,C 180,E1 -8438.415,E2 -8438.415} C_VEL
LIN {X 0,Y 453.527,Z 184.805,A -85,B 0,C 180,E1 -8441.008,E2 -8441.008} C_VEL
LIN {X 0,Y 453.574,Z 184.8,A -85,B 0,C 180,E1 -8443.879,E2 -8443.879} C_VEL
LIN {X 0,Y 453.568,Z 184.803,A -85,B 0,C 180,E1 -8447.471,E2 -8447.471} C_VEL
LIN {X 0,Y 453.589,Z 184.798,A -85,B 0,C 180,E1 -8451.086,E2 -8451.086} C_VEL
LIN {X 0,Y 453.669,Z 184.788,A -85,B 0,C 180,E1 -8453.774,E2 -8453.774} C_VEL
LIN {X 0,Y 453.746,Z 184.779,A -85,B 0,C 180,E1 -8457.336,E2 -8457.336} C_VEL
LIN {X 0,Y 453.825,Z 184.768,A -85,B 0,C 180,E1 -8459.999,E2 -8459.999} C_VEL
LIN {X 0,Y 453.746,Z 184.778,A -85,B 0,C 180,E1 -8462.663,E2 -8462.663} C_VEL
LIN {X 0,Y 453.669,Z 184.786,A -85,B 0,C 180,E1 -8466.225,E2 -8466.225} C_VEL
LIN {X 0,Y 453.588,Z 184.799,A -85,B 0,C 180,E1 -8468.913,E2 -8468.913} C_VEL
LIN {X 0,Y 453.566,Z 184.8,A -85,B 0,C 180,E1 -8472.528,E2 -8472.528} C_VEL
LIN {X 0,Y 453.546,Z 184.802,A -85,B 0,C 180,E1 -8476.195,E2 -8476.195} C_VEL
LIN {X 0,Y 453.518,Z 184.808,A -85,B 0,C 180,E1 -8479.039,E2 -8479.039} C_VEL
LIN {X 0,Y 453.477,Z 184.811,A -85,B 0,C 180,E1 -8481.835,E2 -8481.835} C_VEL
LIN {X 0,Y 453.5,Z 184.809,A -85,B 0,C 180,E1 -8484.734,E2 -8484.734} C_VEL
LIN {X 0,Y 453.537,Z 184.803,A -85,B 0,C 180,E1 -8487.96,E2 -8487.96} C_VEL
LIN {X 0,Y 453.465,Z 184.811,A -85,B 0,C 180,E1 -8491.524,E2 -8491.524} C_VEL
LIN {X 0,Y 453.487,Z 184.81,A -85,B 0,C 180,E1 -8494.777,E2 -8494.777} C_VEL
LIN {X 0,Y 453.47,Z 184.814,A -85,B 0,C 180,E1 -8498.31,E2 -8498.31} C_VEL
LIN {X 0,Y 453.49,Z 184.81,A -85,B 0,C 180,E1 -8500.608,E2 -8500.608} C_VEL
LIN {X 0,Y 453.451,Z 184.813,A -85,B 0,C 180,E1 -8503.243,E2 -8503.243} C_VEL
LIN {X 0,Y 453.461,Z 184.814,A -85,B 0,C 180,E1 -8505.778,E2 -8505.778} C_VEL
LIN {X 0,Y 453.474,Z 184.812,A -85,B 0,C 180,E1 -8508.208,E2 -8508.208} C_VEL
LIN {X 0,Y 453.489,Z 184.808,A -85,B 0,C 180,E1 -8510.792,E2 -8510.792} C_VEL
LIN {X 0,Y 453.451,Z 184.816,A -85,B 0,C 180,E1 -8513.917,E2 -8513.917} C_VEL
LIN {X 0,Y 453.477,Z 184.811,A -85,B 0,C 180,E1 -8517.15,E2 -8517.15} C_VEL
LIN {X 0,Y 453.507,Z 184.807,A -85,B 0,C 180,E1 -8520.27,E2 -8520.27} C_VEL
LIN {X 0,Y 453.502,Z 184.809,A -85,B 0,C 180,E1 -8523.293,E2 -8523.293} C_VEL
LIN {X 0,Y 453.496,Z 184.809,A -85,B 0,C 180,E1 -8526.238,E2 -8526.238} C_VEL
LIN {X 0,Y 453.475,Z 184.813,A -85,B 0,C 180,E1 -8529.117,E2 -8529.117} C_VEL
LIN {X 0,Y 453.503,Z 184.807,A -85,B 0,C 180,E1 -8531.944,E2 -8531.944} C_VEL
LIN {X 0,Y 453.533,Z 184.805,A -85,B 0,C 180,E1 -8534.726,E2 -8534.726} C_VEL
LIN {X 0,Y 453.593,Z 184.797,A -85,B 0,C 180,E1 -8537.472,E2 -8537.472} C_VEL
LIN {X 0,Y 453.584,Z 184.799,A -85,B 0,C 180,E1 -8541.086,E2 -8541.086} C_VEL
LIN {X 0,Y 453.628,Z 184.792,A -85,B 0,C 180,E1 -8543.085,E2 -8543.085} C_VEL
LIN {X 0,Y 452.943,Z 184.876,A -85,B 0,C 180,E1 -8543.826,E2 -8543.826} C_VEL
LIN {X 0,Y 449.996,Z 185.246,A -85,B 0,C 180,E1 -8545.027,E2 -8545.027} C_VEL
LIN {X 0,Y 447.57,Z 185.547,A -85,B 0,C 180,E1 -8545.997,E2 -8545.997} C_VEL
LIN {X 0,Y 446.625,Z 185.666,A -85,B 0,C 180,E1 -8546.747,E2 -8546.747} C_VEL
LIN {X 0,Y 446.6,Z 185.666,A -85,B 0,C 180,E1 -8547.001,E2 -8547.001} C_VEL
LIN {X 0,Y 446.783,Z 185.645,A -85,B 0,C 180,E1 -8550,E2 -8550} C_VEL
LIN {X 0,Y 446.701,Z 185.656,A -85,B 0,C 180,E1 -8552.705,E2 -8552.705} C_VEL
LIN {X 0,Y 446.638,Z 185.665,A -85,B 0,C 180,E1 -8556.324,E2 -8556.324} C_VEL
LIN {X 0,Y 446.53,Z 185.676,A -85,B 0,C 180,E1 -8559.055,E2 -8559.055} C_VEL
LIN {X 0,Y 446.469,Z 185.685,A -85,B 0,C 180,E1 -8562.595,E2 -8562.595} C_VEL
LIN {X 0,Y 446.174,Z 185.913,A -85,B 0,C 180,E1 -8565.064,E2 -8565.064} C_VEL
LIN {X 0,Y 445.995,Z 190.715,A -85,B 0,C 180,E1 -8568.37,E2 -8568.37} C_VEL
LIN {X 0,Y 445.882,Z 195.475,A -85,B 0,C 180,E1 -8571.575,E2 -8571.575} C_VEL
LIN {X 0,Y 445.753,Z 200.93,A -85,B 0,C 180,E1 -8575.195,E2 -8575.195} C_VEL
LIN {X 0,Y 445.601,Z 205.58,A -85,B 0,C 180,E1 -8578.239,E2 -8578.239} C_VEL
LIN {X 0,Y 445.527,Z 210.804,A -85,B 0,C 180,E1 -8581.591,E2 -8581.591} C_VEL
LIN {X 0,Y 445.537,Z 213.791,A -85,B 0,C 180,E1 -8583.375,E2 -8583.375} C_VEL
LIN {X 0,Y 447.243,Z 224.235,A -85,B 0,C 180,E1 -8583.839,E2 -8583.839} C_VEL
LIN {X 0,Y 447.642,Z 228.794,A -85,B 0,C 180,E1 -8584.076,E2 -8584.076} C_VEL
LIN {X 0,Y 447.299,Z 238.469,A -85,B 0,C 180,E1 -8584.701,E2 -8584.701} C_VEL
LIN {X 0,Y 447.034,Z 246.241,A -85,B 0,C 180,E1 -8585.34,E2 -8585.34} C_VEL
LIN {X 0,Y 446.766,Z 252.935,A -85,B 0,C 180,E1 -8586.011,E2 -8586.011} C_VEL
LIN {X 0,Y 446.408,Z 260.111,A -85,B 0,C 180,E1 -8586.885,E2 -8586.885} C_VEL
LIN {X 0,Y 446.116,Z 267.636,A -85,B 0,C 180,E1 -8588.032,E2 -8588.032} C_VEL
LIN {X 0,Y 445.86,Z 272.997,A -85,B 0,C 180,E1 -8589.088,E2 -8589.088} C_VEL
LIN {X 0,Y 445.65,Z 277.723,A -85,B 0,C 180,E1 -8590.284,E2 -8590.284} C_VEL
LIN {X 0,Y 445.515,Z 281.302,A -85,B 0,C 180,E1 -8591.495,E2 -8591.495} C_VEL
LIN {X 0,Y 445.423,Z 283.832,A -85,B 0,C 180,E1 -8592.724,E2 -8592.724} C_VEL
LIN {X 0,Y 445.359,Z 285.338,A -85,B 0,C 180,E1 -8593.975,E2 -8593.975} C_VEL
LIN {X 0,Y 445.33,Z 285.746,A -85,B 0,C 180,E1 -8595.249,E2 -8595.249} C_VEL
LIN {X 0,Y 445.384,Z 285.053,A -85,B 0,C 180,E1 -8596.541,E2 -8596.541} C_VEL
LIN {X 0,Y 445.449,Z 284.237,A -85,B 0,C 180,E1 -8597.281,E2 -8597.281} C_VEL
LIN {X 0,Y 445.519,Z 281.924,A -85,B 0,C 180,E1 -8598.507,E2 -8598.507} C_VEL
LIN {X 0,Y 445.682,Z 278.543,A -85,B 0,C 180,E1 -8599.721,E2 -8599.721} C_VEL
LIN {X 0,Y 445.894,Z 274.046,A -85,B 0,C 180,E1 -8600.917,E2 -8600.917} C_VEL
LIN {X 0,Y 446.206,Z 268.278,A -85,B 0,C 180,E1 -8602.102,E2 -8602.102} C_VEL
LIN {X 0,Y 446.509,Z 260.817,A -85,B 0,C 180,E1 -8603.266,E2 -8603.266} C_VEL
LIN {X 0,Y 446.854,Z 253.81,A -85,B 0,C 180,E1 -8604.138,E2 -8604.138} C_VEL
LIN {X 0,Y 447.204,Z 246.417,A -85,B 0,C 180,E1 -8604.888,E2 -8604.888} C_VEL
LIN {X 0,Y 447.521,Z 237.072,A -85,B 0,C 180,E1 -8605.649,E2 -8605.649} C_VEL
LIN {X 0,Y 447.89,Z 227.977,A -85,B 0,C 180,E1 -8606.204,E2 -8606.204} C_VEL
LIN {X 0,Y 446.285,Z 218.067,A -85,B 0,C 180,E1 -8606.7,E2 -8606.7} C_VEL
LIN {X 0,Y 445.586,Z 214.125,A -85,B 0,C 180,E1 -8606.886,E2 -8606.886} C_VEL
LIN {X 0,Y 445.653,Z 209.185,A -85,B 0,C 180,E1 -8610.153,E2 -8610.153} C_VEL
LIN {X 0,Y 445.736,Z 205.241,A -85,B 0,C 180,E1 -8612.792,E2 -8612.792} C_VEL
LIN {X 0,Y 445.879,Z 200.369,A -85,B 0,C 180,E1 -8616.093,E2 -8616.093} C_VEL
LIN {X 0,Y 446.01,Z 196.502,A -85,B 0,C 180,E1 -8618.752,E2 -8618.752} C_VEL
LIN {X 0,Y 446.143,Z 192.383,A -85,B 0,C 180,E1 -8621.637,E2 -8621.637} C_VEL
LIN {X 0,Y 446.271,Z 188.375,A -85,B 0,C 180,E1 -8624.472,E2 -8624.472} C_VEL
LIN {X 0,Y 446.299,Z 185.792,A -85,B 0,C 180,E1 -8626.338,E2 -8626.338} C_VEL
LIN {X 0,Y 446.504,Z 185.684,A -85,B 0,C 180,E1 -8628.194,E2 -8628.194} C_VEL
LIN {X 0,Y 446.601,Z 185.672,A -85,B 0,C 180,E1 -8631.859,E2 -8631.859} C_VEL
LIN {X 0,Y 446.646,Z 185.668,A -85,B 0,C 180,E1 -8634.583,E2 -8634.583} C_VEL
LIN {X 0,Y 446.667,Z 185.662,A -85,B 0,C 180,E1 -8638.197,E2 -8638.197} C_VEL
LIN {X 0,Y 446.795,Z 185.645,A -85,B 0,C 180,E1 -8640.001,E2 -8640.001} C_VEL
LIN {X 0,Y 446.692,Z 185.657,A -85,B 0,C 180,E1 -8642.706,E2 -8642.706} C_VEL
LIN {X 0,Y 446.643,Z 185.663,A -85,B 0,C 180,E1 -8646.324,E2 -8646.324} C_VEL
LIN {X 0,Y 446.536,Z 185.677,A -85,B 0,C 180,E1 -8649.056,E2 -8649.056} C_VEL
LIN {X 0,Y 446.524,Z 185.68,A -85,B 0,C 180,E1 -8652.73,E2 -8652.73} C_VEL
LIN {X 0,Y 446.499,Z 185.682,A -85,B 0,C 180,E1 -8656.228,E2 -8656.228} C_VEL
LIN {X 0,Y 446.472,Z 185.684,A -85,B 0,C 180,E1 -8659.304,E2 -8659.304} C_VEL
LIN {X 0,Y 446.42,Z 185.692,A -85,B 0,C 180,E1 -8662.2,E2 -8662.2} C_VEL
LIN {X 0,Y 446.446,Z 185.687,A -85,B 0,C 180,E1 -8665.154,E2 -8665.154} C_VEL
LIN {X 0,Y 446.487,Z 185.683,A -85,B 0,C 180,E1 -8668.179,E2 -8668.179} C_VEL
LIN {X 0,Y 446.422,Z 185.69,A -85,B 0,C 180,E1 -8671.775,E2 -8671.775} C_VEL
LIN {X 0,Y 446.431,Z 185.691,A -85,B 0,C 180,E1 -8674.523,E2 -8674.523} C_VEL
LIN {X 0,Y 446.417,Z 185.693,A -85,B 0,C 180,E1 -8678.079,E2 -8678.079} C_VEL
LIN {X 0,Y 446.429,Z 185.691,A -85,B 0,C 180,E1 -8680.918,E2 -8680.918} C_VEL
LIN {X 0,Y 446.404,Z 185.697,A -85,B 0,C 180,E1 -8683.846,E2 -8683.846} C_VEL
LIN {X 0,Y 446.401,Z 185.696,A -85,B 0,C 180,E1 -8686.404,E2 -8686.404} C_VEL
LIN {X 0,Y 446.429,Z 185.691,A -85,B 0,C 180,E1 -8689.083,E2 -8689.083} C_VEL
LIN {X 0,Y 446.418,Z 185.694,A -85,B 0,C 180,E1 -8691.921,E2 -8691.921} C_VEL
LIN {X 0,Y 446.482,Z 185.751,A -85,B 0,C 180,E1 -8694.535,E2 -8694.535} C_VEL
LIN {X 0,Y 447.522,Z 191.374,A -85,B 0,C 180,E1 -8697.194,E2 -8697.194} C_VEL
LIN {X 0,Y 447.959,Z 195.106,A -85,B 0,C 180,E1 -8698.82,E2 -8698.82} C_VEL
LIN {X 0,Y 447.664,Z 200.129,A -85,B 0,C 180,E1 -8700.878,E2 -8700.878} C_VEL
LIN {X 0,Y 447.063,Z 207.758,A -85,B 0,C 180,E1 -8703.885,E2 -8703.885} C_VEL
LIN {X 0,Y 446.619,Z 215.491,A -85,B 0,C 180,E1 -8706.834,E2 -8706.834} C_VEL
LIN {X 0,Y 446.234,Z 224.695,A -85,B 0,C 180,E1 -8710.208,E2 -8710.208} C_VEL
LIN {X 0,Y 445.886,Z 233.964,A -85,B 0,C 180,E1 -8713.518,E2 -8713.518} C_VEL
LIN {X 0,Y 445.667,Z 243.334,A -85,B 0,C 180,E1 -8716.782,E2 -8716.782} C_VEL
LIN {X 0,Y 445.653,Z 244.858,A -85,B 0,C 180,E1 -8717.309,E2 -8717.309} C_VEL
LIN {X 0,Y 446.96,Z 256.596,A -85,B 0,C 180,E1 -8717.735,E2 -8717.735} C_VEL
LIN {X 0,Y 447.484,Z 266.109,A -85,B 0,C 180,E1 -8718.219,E2 -8718.219} C_VEL
LIN {X 0,Y 447.135,Z 276.47,A -85,B 0,C 180,E1 -8718.899,E2 -8718.899} C_VEL
LIN {X 0,Y 446.762,Z 284.646,A -85,B 0,C 180,E1 -8719.578,E2 -8719.578} C_VEL
LIN {X 0,Y 446.415,Z 292.423,A -85,B 0,C 180,E1 -8720.371,E2 -8720.371} C_VEL
LIN {X 0,Y 446.068,Z 300.577,A -85,B 0,C 180,E1 -8721.392,E2 -8721.392} C_VEL
LIN {X 0,Y 445.806,Z 307.724,A -85,B 0,C 180,E1 -8722.527,E2 -8722.527} C_VEL
LIN {X 0,Y 445.578,Z 313.364,A -85,B 0,C 180,E1 -8723.661,E2 -8723.661} C_VEL
LIN {X 0,Y 445.51,Z 318.618,A -85,B 0,C 180,E1 -8725.023,E2 -8725.023} C_VEL
LIN {X 0,Y 445.44,Z 322.479,A -85,B 0,C 180,E1 -8726.382,E2 -8726.382} C_VEL
LIN {X 0,Y 445.459,Z 324.255,A -85,B 0,C 180,E1 -8727.287,E2 -8727.287} C_VEL
LIN {X 0,Y 445.399,Z 325.521,A -85,B 0,C 180,E1 -8728.192,E2 -8728.192} C_VEL
LIN {X 0,Y 445.396,Z 326.305,A -85,B 0,C 180,E1 -8729.096,E2 -8729.096} C_VEL
LIN {X 0,Y 445.405,Z 326.604,A -85,B 0,C 180,E1 -8730,E2 -8730} C_VEL
LIN {X 0,Y 445.396,Z 326.31,A -85,B 0,C 180,E1 -8730.904,E2 -8730.904} C_VEL
LIN {X 0,Y 445.399,Z 325.501,A -85,B 0,C 180,E1 -8731.809,E2 -8731.809} C_VEL
LIN {X 0,Y 445.459,Z 324.207,A -85,B 0,C 180,E1 -8732.713,E2 -8732.713} C_VEL
LIN {X 0,Y 445.412,Z 321.241,A -85,B 0,C 180,E1 -8734.072,E2 -8734.072} C_VEL
LIN {X 0,Y 445.534,Z 316.992,A -85,B 0,C 180,E1 -8735.431,E2 -8735.431} C_VEL
LIN {X 0,Y 445.66,Z 311.083,A -85,B 0,C 180,E1 -8736.792,E2 -8736.792} C_VEL
LIN {X 0,Y 445.826,Z 306.162,A -85,B 0,C 180,E1 -8737.701,E2 -8737.701} C_VEL
LIN {X 0,Y 446.06,Z 300.225,A -85,B 0,C 180,E1 -8738.609,E2 -8738.609} C_VEL
LIN {X 0,Y 446.35,Z 292.99,A -85,B 0,C 180,E1 -8739.516,E2 -8739.516} C_VEL
LIN {X 0,Y 446.662,Z 285.264,A -85,B 0,C 180,E1 -8740.311,E2 -8740.311} C_VEL
LIN {X 0,Y 447.05,Z 277.146,A -85,B 0,C 180,E1 -8740.989,E2 -8740.989} C_VEL
LIN {X 0,Y 447.327,Z 268.713,A -85,B 0,C 180,E1 -8741.556,E2 -8741.556} C_VEL
LIN {X 0,Y 447.376,Z 262.909,A -85,B 0,C 180,E1 -8741.878,E2 -8741.878} C_VEL
LIN {X 0,Y 446.508,Z 253.079,A -85,B 0,C 180,E1 -8742.321,E2 -8742.321} C_VEL
LIN {X 0,Y 445.649,Z 245.354,A -85,B 0,C 180,E1 -8742.581,E2 -8742.581} C_VEL
LIN {X 0,Y 445.889,Z 235.672,A -85,B 0,C 180,E1 -8745.956,E2 -8745.956} C_VEL
LIN {X 0,Y 446.189,Z 226.181,A -85,B 0,C 180,E1 -8749.316,E2 -8749.316} C_VEL
LIN {X 0,Y 446.589,Z 216.871,A -85,B 0,C 180,E1 -8752.679,E2 -8752.679} C_VEL
LIN {X 0,Y 447.096,Z 207.564,A -85,B 0,C 180,E1 -8756.113,E2 -8756.113} C_VEL
LIN {X 0,Y 447.613,Z 199.641,A -85,B 0,C 180,E1 -8759.126,E2 -8759.126} C_VEL
LIN {X 0,Y 447.875,Z 194.379,A -85,B 0,C 180,E1 -8761.187,E2 -8761.187} C_VEL
LIN {X 0,Y 446.828,Z 187.695,A -85,B 0,C 180,E1 -8763.985,E2 -8763.985} C_VEL
LIN {X 0,Y 446.475,Z 185.686,A -85,B 0,C 180,E1 -8764.923,E2 -8764.923} C_VEL
LIN {X 0,Y 446.418,Z 185.692,A -85,B 0,C 180,E1 -8768.079,E2 -8768.079} C_VEL
LIN {X 0,Y 446.43,Z 185.689,A -85,B 0,C 180,E1 -8770.918,E2 -8770.918} C_VEL
LIN {X 0,Y 446.403,Z 185.691,A -85,B 0,C 180,E1 -8773.846,E2 -8773.846} C_VEL
LIN {X 0,Y 446.401,Z 185.694,A -85,B 0,C 180,E1 -8776.404,E2 -8776.404} C_VEL
LIN {X 0,Y 446.426,Z 185.689,A -85,B 0,C 180,E1 -8779.083,E2 -8779.083} C_VEL
LIN {X 0,Y 446.411,Z 185.693,A -85,B 0,C 180,E1 -8782.121,E2 -8782.121} C_VEL
LIN {X 0,Y 446.433,Z 185.687,A -85,B 0,C 180,E1 -8785.477,E2 -8785.477} C_VEL
LIN {X 0,Y 446.42,Z 185.689,A -85,B 0,C 180,E1 -8788.699,E2 -8788.699} C_VEL
LIN {X 0,Y 446.489,Z 185.683,A -85,B 0,C 180,E1 -8791.821,E2 -8791.821} C_VEL
LIN {X 0,Y 446.449,Z 185.686,A -85,B 0,C 180,E1 -8794.847,E2 -8794.847} C_VEL
LIN {X 0,Y 446.453,Z 185.688,A -85,B 0,C 180,E1 -8798.245,E2 -8798.245} C_VEL
LIN {X 0,Y 446.457,Z 185.687,A -85,B 0,C 180,E1 -8801.649,E2 -8801.649} C_VEL
LIN {X 0,Y 446.513,Z 185.678,A -85,B 0,C 180,E1 -8804.479,E2 -8804.479} C_VEL
LIN {X 0,Y 446.522,Z 185.678,A -85,B 0,C 180,E1 -8808.193,E2 -8808.193} C_VEL
LIN {X 0,Y 446.536,Z 185.675,A -85,B 0,C 180,E1 -8810.944,E2 -8810.944} C_VEL
LIN {X 0,Y 446.638,Z 185.665,A -85,B 0,C 180,E1 -8813.675,E2 -8813.675} C_VEL
LIN {X 0,Y 446.693,Z 185.658,A -85,B 0,C 180,E1 -8817.294,E2 -8817.294} C_VEL
LIN {X 0,Y 446.795,Z 185.643,A -85,B 0,C 180,E1 -8819.999,E2 -8819.999} C_VEL
LIN {X 0,Y 446.694,Z 185.657,A -85,B 0,C 180,E1 -8822.705,E2 -8822.705} C_VEL
LIN {X 0,Y 446.638,Z 185.662,A -85,B 0,C 180,E1 -8826.323,E2 -8826.323} C_VEL
LIN {X 0,Y 446.535,Z 185.679,A -85,B 0,C 180,E1 -8829.055,E2 -8829.055} C_VEL
LIN {X 0,Y 446.524,Z 185.679,A -85,B 0,C 180,E1 -8832.729,E2 -8832.729} C_VEL
LIN {X 0,Y 446.497,Z 185.68,A -85,B 0,C 180,E1 -8836.226,E2 -8836.226} C_VEL
LIN {X 0,Y 446.469,Z 185.684,A -85,B 0,C 180,E1 -8839.302,E2 -8839.302} C_VEL
LIN {X 0,Y 446.418,Z 185.692,A -85,B 0,C 180,E1 -8842.198,E2 -8842.198} C_VEL
LIN {X 0,Y 446.444,Z 185.687,A -85,B 0,C 180,E1 -8845.152,E2 -8845.152} C_VEL
LIN {X 0,Y 446.484,Z 185.684,A -85,B 0,C 180,E1 -8848.178,E2 -8848.178} C_VEL
LIN {X 0,Y 446.418,Z 185.69,A -85,B 0,C 180,E1 -8851.774,E2 -8851.774} C_VEL
LIN {X 0,Y 446.429,Z 185.691,A -85,B 0,C 180,E1 -8854.522,E2 -8854.522} C_VEL
LIN {X 0,Y 446.427,Z 185.69,A -85,B 0,C 180,E1 -8858.081,E2 -8858.081} C_VEL
LIN {X 0,Y 446.423,Z 185.69,A -85,B 0,C 180,E1 -8860.916,E2 -8860.916} C_VEL
LIN {X 0,Y 446.397,Z 185.695,A -85,B 0,C 180,E1 -8863.845,E2 -8863.845} C_VEL
LIN {X 0,Y 446.394,Z 185.693,A -85,B 0,C 180,E1 -8866.402,E2 -8866.402} C_VEL
LIN {X 0,Y 446.422,Z 185.69,A -85,B 0,C 180,E1 -8869.081,E2 -8869.081} C_VEL
LIN {X 0,Y 446.422,Z 185.691,A -85,B 0,C 180,E1 -8872.122,E2 -8872.122} C_VEL
LIN {X 0,Y 446.425,Z 185.691,A -85,B 0,C 180,E1 -8875.476,E2 -8875.476} C_VEL
LIN {X 0,Y 446.413,Z 185.69,A -85,B 0,C 180,E1 -8878.699,E2 -8878.699} C_VEL
LIN {X 0,Y 446.477,Z 185.684,A -85,B 0,C 180,E1 -8881.821,E2 -8881.821} C_VEL
LIN {X 0,Y 446.45,Z 185.686,A -85,B 0,C 180,E1 -8884.847,E2 -8884.847} C_VEL
LIN {X 0,Y 446.44,Z 185.686,A -85,B 0,C 180,E1 -8888.244,E2 -8888.244} C_VEL
LIN {X 0,Y 446.449,Z 185.688,A -85,B 0,C 180,E1 -8891.649,E2 -8891.649} C_VEL
LIN {X 0,Y 446.5,Z 185.681,A -85,B 0,C 180,E1 -8894.479,E2 -8894.479} C_VEL
LIN {X 0,Y 446.537,Z 185.675,A -85,B 0,C 180,E1 -8898.193,E2 -8898.193} C_VEL
LIN {X 0,Y 446.591,Z 185.669,A -85,B 0,C 180,E1 -8901.857,E2 -8901.857} C_VEL
LIN {X 0,Y 446.637,Z 185.665,A -85,B 0,C 180,E1 -8904.582,E2 -8904.582} C_VEL
LIN {X 0,Y 446.6,Z 185.666,A -85,B 0,C 180,E1 -8907.001,E2 -8907.001} C_VEL
LIN {X 0,Y 446.075,Z 185.734,A -85,B 0,C 180,E1 -8907.754,E2 -8907.754} C_VEL
LIN {X 0,Y 443.264,Z 186.09,A -85,B 0,C 180,E1 -8908.977,E2 -8908.977} C_VEL
LIN {X 0,Y 440.79,Z 186.398,A -85,B 0,C 180,E1 -8909.964,E2 -8909.964} C_VEL
LIN {X 0,Y 439.706,Z 186.53,A -85,B 0,C 180,E1 -8910.728,E2 -8910.728} C_VEL
LIN {X 0,Y 439.613,Z 186.539,A -85,B 0,C 180,E1 -8910.987,E2 -8910.987} C_VEL
LIN {X 0,Y 439.648,Z 186.535,A -85,B 0,C 180,E1 -8912.749,E2 -8912.749} C_VEL
LIN {X 0,Y 439.61,Z 186.54,A -85,B 0,C 180,E1 -8916.425,E2 -8916.425} C_VEL
LIN {X 0,Y 439.492,Z 186.553,A -85,B 0,C 180,E1 -8919.202,E2 -8919.202} C_VEL
LIN {X 0,Y 439.411,Z 186.564,A -85,B 0,C 180,E1 -8922.678,E2 -8922.678} C_VEL
LIN {X 0,Y 439.117,Z 186.741,A -85,B 0,C 180,E1 -8925.075,E2 -8925.075} C_VEL
LIN {X 0,Y 438.944,Z 191.935,A -85,B 0,C 180,E1 -8928.676,E2 -8928.676} C_VEL
LIN {X 0,Y 438.804,Z 196.416,A -85,B 0,C 180,E1 -8931.733,E2 -8931.733} C_VEL
LIN {X 0,Y 438.682,Z 200.713,A -85,B 0,C 180,E1 -8934.616,E2 -8934.616} C_VEL
LIN {X 0,Y 438.572,Z 205.338,A -85,B 0,C 180,E1 -8937.692,E2 -8937.692} C_VEL
LIN {X 0,Y 438.444,Z 210.183,A -85,B 0,C 180,E1 -8940.86,E2 -8940.86} C_VEL
LIN {X 0,Y 438.423,Z 213.777,A -85,B 0,C 180,E1 -8943.173,E2 -8943.173} C_VEL
LIN {X 0,Y 440.15,Z 224.369,A -85,B 0,C 180,E1 -8943.661,E2 -8943.661} C_VEL
LIN {X 0,Y 440.665,Z 229.389,A -85,B 0,C 180,E1 -8943.931,E2 -8943.931} C_VEL
LIN {X 0,Y 440.281,Z 239.624,A -85,B 0,C 180,E1 -8944.615,E2 -8944.615} C_VEL
LIN {X 0,Y 440.006,Z 247.262,A -85,B 0,C 180,E1 -8945.266,E2 -8945.266} C_VEL
LIN {X 0,Y 439.705,Z 254.625,A -85,B 0,C 180,E1 -8946.037,E2 -8946.037} C_VEL
LIN {X 0,Y 439.266,Z 263.035,A -85,B 0,C 180,E1 -8947.134,E2 -8947.134} C_VEL
LIN {X 0,Y 439.04,Z 268.889,A -85,B 0,C 180,E1 -8948.114,E2 -8948.114} C_VEL
LIN {X 0,Y 438.777,Z 274.079,A -85,B 0,C 180,E1 -8949.191,E2 -8949.191} C_VEL
LIN {X 0,Y 438.604,Z 277.835,A -85,B 0,C 180,E1 -8950.162,E2 -8950.162} C_VEL
LIN {X 0,Y 438.422,Z 282.254,A -85,B 0,C 180,E1 -8951.701,E2 -8951.701} C_VEL
LIN {X 0,Y 438.362,Z 283.763,A -85,B 0,C 180,E1 -8952.484,E2 -8952.484} C_VEL
LIN {X 0,Y 438.277,Z 285.511,A -85,B 0,C 180,E1 -8953.815,E2 -8953.815} C_VEL
LIN {X 0,Y 438.242,Z 286.102,A -85,B 0,C 180,E1 -8955.122,E2 -8955.122} C_VEL
LIN {X 0,Y 438.297,Z 285.554,A -85,B 0,C 180,E1 -8956.411,E2 -8956.411} C_VEL
LIN {X 0,Y 438.37,Z 283.984,A -85,B 0,C 180,E1 -8957.676,E2 -8957.676} C_VEL
LIN {X 0,Y 438.469,Z 281.416,A -85,B 0,C 180,E1 -8958.917,E2 -8958.917} C_VEL
LIN {X 0,Y 438.702,Z 277.406,A -85,B 0,C 180,E1 -8960.26,E2 -8960.26} C_VEL
LIN {X 0,Y 439.032,Z 271.484,A -85,B 0,C 180,E1 -8961.664,E2 -8961.664} C_VEL
LIN {X 0,Y 439.269,Z 266.688,A -85,B 0,C 180,E1 -8962.558,E2 -8962.558} C_VEL
LIN {X 0,Y 439.501,Z 261.108,A -85,B 0,C 180,E1 -8963.42,E2 -8963.42} C_VEL
LIN {X 0,Y 439.852,Z 255.091,A -85,B 0,C 180,E1 -8964.191,E2 -8964.191} C_VEL
LIN {X 0,Y 440.148,Z 248.314,A -85,B 0,C 180,E1 -8964.914,E2 -8964.914} C_VEL
LIN {X 0,Y 440.487,Z 239.739,A -85,B 0,C 180,E1 -8965.654,E2 -8965.654} C_VEL
LIN {X 0,Y 440.885,Z 231.093,A -85,B 0,C 180,E1 -8966.238,E2 -8966.238} C_VEL
LIN {X 0,Y 440.768,Z 226.889,A -85,B 0,C 180,E1 -8966.477,E2 -8966.477} C_VEL
LIN {X 0,Y 439.063,Z 217.418,A -85,B 0,C 180,E1 -8966.954,E2 -8966.954} C_VEL
LIN {X 0,Y 438.488,Z 214.425,A -85,B 0,C 180,E1 -8967.1,E2 -8967.1} C_VEL
LIN {X 0,Y 438.594,Z 209.775,A -85,B 0,C 180,E1 -8970.217,E2 -8970.217} C_VEL
LIN {X 0,Y 438.704,Z 205.138,A -85,B 0,C 180,E1 -8973.35,E2 -8973.35} C_VEL
LIN {X 0,Y 438.85,Z 200.736,A -85,B 0,C 180,E1 -8976.4,E2 -8976.4} C_VEL
LIN {X 0,Y 438.958,Z 196.452,A -85,B 0,C 180,E1 -8979.377,E2 -8979.377} C_VEL
LIN {X 0,Y 439.12,Z 192.353,A -85,B 0,C 180,E1 -8982.298,E2 -8982.298} C_VEL
LIN {X 0,Y 439.236,Z 188.374,A -85,B 0,C 180,E1 -8985.168,E2 -8985.168} C_VEL
LIN {X 0,Y 439.274,Z 187.089,A -85,B 0,C 180,E1 -8986.115,E2 -8986.115} C_VEL
LIN {X 0,Y 439.42,Z 186.57,A -85,B 0,C 180,E1 -8987.323,E2 -8987.323} C_VEL
LIN {X 0,Y 439.5,Z 186.554,A -85,B 0,C 180,E1 -8990.799,E2 -8990.799} C_VEL
LIN {X 0,Y 439.619,Z 186.544,A -85,B 0,C 180,E1 -8993.576,E2 -8993.576} C_VEL
LIN {X 0,Y 439.642,Z 186.537,A -85,B 0,C 180,E1 -8997.252,E2 -8997.252} C_VEL
LIN {X 0,Y 439.765,Z 186.521,A -85,B 0,C 180,E1 -9000.001,E2 -9000.001} C_VEL
LIN {X 0,Y 439.642,Z 186.535,A -85,B 0,C 180,E1 -9002.75,E2 -9002.75} C_VEL
LIN {X 0,Y 439.615,Z 186.538,A -85,B 0,C 180,E1 -9006.426,E2 -9006.426} C_VEL
LIN {X 0,Y 439.499,Z 186.554,A -85,B 0,C 180,E1 -9009.202,E2 -9009.202} C_VEL
LIN {X 0,Y 439.468,Z 186.558,A -85,B 0,C 180,E1 -9012.938,E2 -9012.938} C_VEL
LIN {X 0,Y 439.45,Z 186.561,A -85,B 0,C 180,E1 -9016.349,E2 -9016.349} C_VEL
LIN {X 0,Y 439.405,Z 186.566,A -85,B 0,C 180,E1 -9019.627,E2 -9019.627} C_VEL
LIN {X 0,Y 439.366,Z 186.569,A -85,B 0,C 180,E1 -9022.576,E2 -9022.576} C_VEL
LIN {X 0,Y 439.4,Z 186.564,A -85,B 0,C 180,E1 -9025.586,E2 -9025.586} C_VEL
LIN {X 0,Y 439.42,Z 186.564,A -85,B 0,C 180,E1 -9028.674,E2 -9028.674} C_VEL
LIN {X 0,Y 439.373,Z 186.569,A -85,B 0,C 180,E1 -9032.031,E2 -9032.031} C_VEL
LIN {X 0,Y 439.397,Z 186.565,A -85,B 0,C 180,E1 -9035.341,E2 -9035.341} C_VEL
LIN {X 0,Y 439.379,Z 186.568,A -85,B 0,C 180,E1 -9038.596,E2 -9038.596} C_VEL
LIN {X 0,Y 439.39,Z 186.569,A -85,B 0,C 180,E1 -9041.257,E2 -9041.257} C_VEL
LIN {X 0,Y 439.404,Z 186.568,A -85,B 0,C 180,E1 -9044.729,E2 -9044.729} C_VEL
LIN {X 0,Y 439.398,Z 186.567,A -85,B 0,C 180,E1 -9047.796,E2 -9047.796} C_VEL
LIN {X 0,Y 439.432,Z 186.562,A -85,B 0,C 180,E1 -9050.228,E2 -9050.228} C_VEL
LIN {X 0,Y 439.398,Z 186.6,A -85,B 0,C 180,E1 -9054.217,E2 -9054.217} C_VEL
LIN {X 0,Y 440.548,Z 192.664,A -85,B 0,C 180,E1 -9057.153,E2 -9057.153} C_VEL
LIN {X 0,Y 440.978,Z 196.353,A -85,B 0,C 180,E1 -9058.804,E2 -9058.804} C_VEL
LIN {X 0,Y 440.53,Z 202.607,A -85,B 0,C 180,E1 -9061.406,E2 -9061.406} C_VEL
LIN {X 0,Y 439.943,Z 210.229,A -85,B 0,C 180,E1 -9064.449,E2 -9064.449} C_VEL
LIN {X 0,Y 439.514,Z 217.991,A -85,B 0,C 180,E1 -9067.433,E2 -9067.433} C_VEL
LIN {X 0,Y 439.121,Z 226.983,A -85,B 0,C 180,E1 -9070.783,E2 -9070.783} C_VEL
LIN {X 0,Y 438.743,Z 237.756,A -85,B 0,C 180,E1 -9074.674,E2 -9074.674} C_VEL
LIN {X 0,Y 438.567,Z 244.57,A -85,B 0,C 180,E1 -9077.088,E2 -9077.088} C_VEL
LIN {X 0,Y 439.923,Z 256.263,A -85,B 0,C 180,E1 -9077.525,E2 -9077.525} C_VEL
LIN {X 0,Y 440.547,Z 265.938,A -85,B 0,C 180,E1 -9078.031,E2 -9078.031} C_VEL
LIN {X 0,Y 440.174,Z 276.26,A -85,B 0,C 180,E1 -9078.721,E2 -9078.721} C_VEL
LIN {X 0,Y 439.76,Z 284.411,A -85,B 0,C 180,E1 -9079.41,E2 -9079.41} C_VEL
LIN {X 0,Y 439.411,Z 292.169,A -85,B 0,C 180,E1 -9080.216,E2 -9080.216} C_VEL
LIN {X 0,Y 439.033,Z 300.312,A -85,B 0,C 180,E1 -9081.253,E2 -9081.253} C_VEL
LIN {X 0,Y 438.733,Z 307.441,A -85,B 0,C 180,E1 -9082.406,E2 -9082.406} C_VEL
LIN {X 0,Y 438.506,Z 313.075,A -85,B 0,C 180,E1 -9083.559,E2 -9083.559} C_VEL
LIN {X 0,Y 438.43,Z 316.777,A -85,B 0,C 180,E1 -9084.481,E2 -9084.481} C_VEL
LIN {X 0,Y 438.364,Z 319.813,A -85,B 0,C 180,E1 -9085.402,E2 -9085.402} C_VEL
LIN {X 0,Y 438.336,Z 322.175,A -85,B 0,C 180,E1 -9086.323,E2 -9086.323} C_VEL
LIN {X 0,Y 438.385,Z 323.946,A -85,B 0,C 180,E1 -9087.243,E2 -9087.243} C_VEL
LIN {X 0,Y 438.319,Z 325.205,A -85,B 0,C 180,E1 -9088.162,E2 -9088.162} C_VEL
LIN {X 0,Y 438.306,Z 325.982,A -85,B 0,C 180,E1 -9089.081,E2 -9089.081} C_VEL
LIN {X 0,Y 438.313,Z 326.276,A -85,B 0,C 180,E1 -9090,E2 -9090} C_VEL
LIN {X 0,Y 438.306,Z 325.981,A -85,B 0,C 180,E1 -9090.919,E2 -9090.919} C_VEL
LIN {X 0,Y 438.319,Z 325.163,A -85,B 0,C 180,E1 -9091.838,E2 -9091.838} C_VEL
LIN {X 0,Y 438.386,Z 323.861,A -85,B 0,C 180,E1 -9092.757,E2 -9092.757} C_VEL
LIN {X 0,Y 438.323,Z 320.883,A -85,B 0,C 180,E1 -9094.138,E2 -9094.138} C_VEL
LIN {X 0,Y 438.43,Z 316.618,A -85,B 0,C 180,E1 -9095.519,E2 -9095.519} C_VEL
LIN {X 0,Y 438.603,Z 310.679,A -85,B 0,C 180,E1 -9096.903,E2 -9096.903} C_VEL
LIN {X 0,Y 438.766,Z 305.739,A -85,B 0,C 180,E1 -9097.825,E2 -9097.825} C_VEL
LIN {X 0,Y 439.03,Z 299.778,A -85,B 0,C 180,E1 -9098.747,E2 -9098.747} C_VEL
LIN {X 0,Y 439.317,Z 292.512,A -85,B 0,C 180,E1 -9099.67,E2 -9099.67} C_VEL
LIN {X 0,Y 439.64,Z 284.747,A -85,B 0,C 180,E1 -9100.477,E2 -9100.477} C_VEL
LIN {X 0,Y 440.06,Z 276.582,A -85,B 0,C 180,E1 -9101.166,E2 -9101.166} C_VEL
LIN {X 0,Y 440.411,Z 266.222,A -85,B 0,C 180,E1 -9101.856,E2 -9101.856} C_VEL
LIN {X 0,Y 439.6,Z 254.562,A -85,B 0,C 180,E1 -9102.432,E2 -9102.432} C_VEL
LIN {X 0,Y 438.549,Z 245.089,A -85,B 0,C 180,E1 -9102.768,E2 -9102.768} C_VEL
LIN {X 0,Y 438.809,Z 235.831,A -85,B 0,C 180,E1 -9106.061,E2 -9106.061} C_VEL
LIN {X 0,Y 439.175,Z 225.937,A -85,B 0,C 180,E1 -9109.637,E2 -9109.637} C_VEL
LIN {X 0,Y 439.58,Z 216.645,A -85,B 0,C 180,E1 -9113.061,E2 -9113.061} C_VEL
LIN {X 0,Y 440.041,Z 208.698,A -85,B 0,C 180,E1 -9116.054,E2 -9116.054} C_VEL
LIN {X 0,Y 440.581,Z 200.803,A -85,B 0,C 180,E1 -9119.112,E2 -9119.112} C_VEL
LIN {X 0,Y 440.87,Z 195.526,A -85,B 0,C 180,E1 -9121.204,E2 -9121.204} C_VEL
LIN {X 0,Y 439.854,Z 188.949,A -85,B 0,C 180,E1 -9124.003,E2 -9124.003} C_VEL
LIN {X 0,Y 439.396,Z 186.567,A -85,B 0,C 180,E1 -9125.087,E2 -9125.087} C_VEL
LIN {X 0,Y 439.381,Z 186.568,A -85,B 0,C 180,E1 -9128.596,E2 -9128.596} C_VEL
LIN {X 0,Y 439.392,Z 186.565,A -85,B 0,C 180,E1 -9131.257,E2 -9131.257} C_VEL
LIN {X 0,Y 439.403,Z 186.565,A -85,B 0,C 180,E1 -9134.729,E2 -9134.729} C_VEL
LIN {X 0,Y 439.388,Z 186.565,A -85,B 0,C 180,E1 -9137.794,E2 -9137.794} C_VEL
LIN {X 0,Y 439.362,Z 186.571,A -85,B 0,C 180,E1 -9140.22,E2 -9140.22} C_VEL
LIN {X 0,Y 439.378,Z 186.568,A -85,B 0,C 180,E1 -9143.713,E2 -9143.713} C_VEL
LIN {X 0,Y 439.377,Z 186.567,A -85,B 0,C 180,E1 -9147.054,E2 -9147.054} C_VEL
LIN {X 0,Y 439.386,Z 186.567,A -85,B 0,C 180,E1 -9150.274,E2 -9150.274} C_VEL
LIN {X 0,Y 439.432,Z 186.561,A -85,B 0,C 180,E1 -9153.396,E2 -9153.396} C_VEL
LIN {X 0,Y 439.389,Z 186.565,A -85,B 0,C 180,E1 -9156.429,E2 -9156.429} C_VEL
LIN {X 0,Y 439.393,Z 186.566,A -85,B 0,C 180,E1 -9159.397,E2 -9159.397} C_VEL
LIN {X 0,Y 439.431,Z 186.561,A -85,B 0,C 180,E1 -9162.309,E2 -9162.309} C_VEL
LIN {X 0,Y 439.452,Z 186.56,A -85,B 0,C 180,E1 -9165.173,E2 -9165.173} C_VEL
LIN {X 0,Y 439.488,Z 186.554,A -85,B 0,C 180,E1 -9168.001,E2 -9168.001} C_VEL
LIN {X 0,Y 439.508,Z 186.552,A -85,B 0,C 180,E1 -9171.725,E2 -9171.725} C_VEL
LIN {X 0,Y 439.619,Z 186.536,A -85,B 0,C 180,E1 -9174.495,E2 -9174.495} C_VEL
LIN {X 0,Y 439.636,Z 186.533,A -85,B 0,C 180,E1 -9178.167,E2 -9178.167} C_VEL
LIN {X 0,Y 439.764,Z 186.519,A -85,B 0,C 180,E1 -9179.999,E2 -9179.999} C_VEL
LIN {X 0,Y 439.643,Z 186.535,A -85,B 0,C 180,E1 -9182.748,E2 -9182.748} C_VEL
LIN {X 0,Y 439.608,Z 186.538,A -85,B 0,C 180,E1 -9186.425,E2 -9186.425} C_VEL
LIN {X 0,Y 439.498,Z 186.554,A -85,B 0,C 180,E1 -9189.201,E2 -9189.201} C_VEL
LIN {X 0,Y 439.468,Z 186.559,A -85,B 0,C 180,E1 -9192.937,E2 -9192.937} C_VEL
LIN {X 0,Y 439.448,Z 186.559,A -85,B 0,C 180,E1 -9196.347,E2 -9196.347} C_VEL
LIN {X 0,Y 439.403,Z 186.563,A -85,B 0,C 180,E1 -9199.625,E2 -9199.625} C_VEL
LIN {X 0,Y 439.364,Z 186.57,A -85,B 0,C 180,E1 -9202.574,E2 -9202.574} C_VEL
LIN {X 0,Y 439.397,Z 186.564,A -85,B 0,C 180,E1 -9205.584,E2 -9205.584} C_VEL
LIN {X 0,Y 439.417,Z 186.563,A -85,B 0,C 180,E1 -9208.672,E2 -9208.672} C_VEL
LIN {X 0,Y 439.369,Z 186.57,A -85,B 0,C 180,E1 -9212.029,E2 -9212.029} C_VEL
LIN {X 0,Y 439.394,Z 186.564,A -85,B 0,C 180,E1 -9215.34,E2 -9215.34} C_VEL
LIN {X 0,Y 439.38,Z 186.567,A -85,B 0,C 180,E1 -9218.594,E2 -9218.594} C_VEL
LIN {X 0,Y 439.385,Z 186.566,A -85,B 0,C 180,E1 -9221.256,E2 -9221.256} C_VEL
LIN {X 0,Y 439.397,Z 186.565,A -85,B 0,C 180,E1 -9224.728,E2 -9224.728} C_VEL
LIN {X 0,Y 439.391,Z 186.567,A -85,B 0,C 180,E1 -9227.795,E2 -9227.795} C_VEL
LIN {X 0,Y 439.42,Z 186.562,A -85,B 0,C 180,E1 -9230.226,E2 -9230.226} C_VEL
LIN {X 0,Y 439.371,Z 186.57,A -85,B 0,C 180,E1 -9233.712,E2 -9233.712} C_VEL
LIN {X 0,Y 439.366,Z 186.569,A -85,B 0,C 180,E1 -9237.053,E2 -9237.053} C_VEL
LIN {X 0,Y 439.39,Z 186.565,A -85,B 0,C 180,E1 -9240.274,E2 -9240.274} C_VEL
LIN {X 0,Y 439.426,Z 186.563,A -85,B 0,C 180,E1 -9243.588,E2 -9243.588} C_VEL
LIN {X 0,Y 439.379,Z 186.566,A -85,B 0,C 180,E1 -9246.429,E2 -9246.429} C_VEL
LIN {X 0,Y 439.381,Z 186.568,A -85,B 0,C 180,E1 -9249.397,E2 -9249.397} C_VEL
LIN {X 0,Y 439.423,Z 186.56,A -85,B 0,C 180,E1 -9252.309,E2 -9252.309} C_VEL
LIN {X 0,Y 439.443,Z 186.561,A -85,B 0,C 180,E1 -9255.174,E2 -9255.174} C_VEL
LIN {X 0,Y 439.503,Z 186.551,A -85,B 0,C 180,E1 -9258.002,E2 -9258.002} C_VEL
LIN {X 0,Y 439.539,Z 186.547,A -85,B 0,C 180,E1 -9261.726,E2 -9261.726} C_VEL
LIN {X 0,Y 439.613,Z 186.539,A -85,B 0,C 180,E1 -9264.495,E2 -9264.495} C_VEL
LIN {X 0,Y 439.625,Z 186.536,A -85,B 0,C 180,E1 -9268.168,E2 -9268.168} C_VEL
LIN {X 0,Y 439.753,Z 186.52,A -85,B 0,C 180,E1 -9270,E2 -9270} C_VEL
LIN {X 0,Y 439.613,Z 186.539,A -85,B 0,C 180,E1 -9270.987,E2 -9270.987} C_VEL
LIN {X 0,Y 438.896,Z 186.626,A -85,B 0,C 180,E1 -9271.751,E2 -9271.751} C_VEL
LIN {X 0,Y 435.917,Z 187,A -85,B 0,C 180,E1 -9272.99,E2 -9272.99} C_VEL
LIN {X 0,Y 433.466,Z 187.307,A -85,B 0,C 180,E1 -9273.99,E2 -9273.99} C_VEL
LIN {X 0,Y 432.493,Z 187.427,A -85,B 0,C 180,E1 -9274.765,E2 -9274.765} C_VEL
LIN {X 0,Y 432.456,Z 187.429,A -85,B 0,C 180,E1 -9275.027,E2 -9275.027} C_VEL
LIN {X 0,Y 432.577,Z 187.414,A -85,B 0,C 180,E1 -9277.679,E2 -9277.679} C_VEL
LIN {X 0,Y 432.378,Z 187.438,A -85,B 0,C 180,E1 -9281.248,E2 -9281.248} C_VEL
LIN {X 0,Y 432.308,Z 187.447,A -85,B 0,C 180,E1 -9283.155,E2 -9283.155} C_VEL
LIN {X 0,Y 432.077,Z 187.578,A -85,B 0,C 180,E1 -9285.085,E2 -9285.085} C_VEL
LIN {X 0,Y 431.884,Z 191.727,A -85,B 0,C 180,E1 -9288.01,E2 -9288.01} C_VEL
LIN {X 0,Y 431.753,Z 196.042,A -85,B 0,C 180,E1 -9290.984,E2 -9290.984} C_VEL
LIN {X 0,Y 431.641,Z 200.823,A -85,B 0,C 180,E1 -9294.249,E2 -9294.249} C_VEL
LIN {X 0,Y 431.514,Z 205.132,A -85,B 0,C 180,E1 -9297.131,E2 -9297.131} C_VEL
LIN {X 0,Y 431.394,Z 209.956,A -85,B 0,C 180,E1 -9300.333,E2 -9300.333} C_VEL
LIN {X 0,Y 431.342,Z 214,A -85,B 0,C 180,E1 -9302.977,E2 -9302.977} C_VEL
LIN {X 0,Y 433.362,Z 226.411,A -85,B 0,C 180,E1 -9303.581,E2 -9303.581} C_VEL
LIN {X 0,Y 433.668,Z 230.153,A -85,B 0,C 180,E1 -9303.793,E2 -9303.793} C_VEL
LIN {X 0,Y 433.343,Z 238.752,A -85,B 0,C 180,E1 -9304.368,E2 -9304.368} C_VEL
LIN {X 0,Y 433.047,Z 246.676,A -85,B 0,C 180,E1 -9305.037,E2 -9305.037} C_VEL
LIN {X 0,Y 432.715,Z 253.859,A -85,B 0,C 180,E1 -9305.782,E2 -9305.782} C_VEL
LIN {X 0,Y 432.339,Z 260.979,A -85,B 0,C 180,E1 -9306.684,E2 -9306.684} C_VEL
LIN {X 0,Y 432.014,Z 268.7,A -85,B 0,C 180,E1 -9307.917,E2 -9307.917} C_VEL
LIN {X 0,Y 431.736,Z 273.914,A -85,B 0,C 180,E1 -9308.994,E2 -9308.994} C_VEL
LIN {X 0,Y 431.545,Z 278.019,A -85,B 0,C 180,E1 -9310.057,E2 -9310.057} C_VEL
LIN {X 0,Y 431.386,Z 281.064,A -85,B 0,C 180,E1 -9311.058,E2 -9311.058} C_VEL
LIN {X 0,Y 431.308,Z 283.135,A -85,B 0,C 180,E1 -9311.919,E2 -9311.919} C_VEL
LIN {X 0,Y 431.239,Z 285.178,A -85,B 0,C 180,E1 -9313.195,E2 -9313.195} C_VEL
LIN {X 0,Y 431.149,Z 286.225,A -85,B 0,C 180,E1 -9314.501,E2 -9314.501} C_VEL
LIN {X 0,Y 431.159,Z 286.232,A -85,B 0,C 180,E1 -9315.825,E2 -9315.825} C_VEL
LIN {X 0,Y 431.267,Z 285.163,A -85,B 0,C 180,E1 -9317.166,E2 -9317.166} C_VEL
LIN {X 0,Y 431.365,Z 282.85,A -85,B 0,C 180,E1 -9318.543,E2 -9318.543} C_VEL
LIN {X 0,Y 431.562,Z 279.087,A -85,B 0,C 180,E1 -9319.942,E2 -9319.942} C_VEL
LIN {X 0,Y 431.805,Z 275.231,A -85,B 0,C 180,E1 -9321.011,E2 -9321.011} C_VEL
LIN {X 0,Y 432.067,Z 270.345,A -85,B 0,C 180,E1 -9322.084,E2 -9322.084} C_VEL
LIN {X 0,Y 432.444,Z 263.19,A -85,B 0,C 180,E1 -9323.328,E2 -9323.328} C_VEL
LIN {X 0,Y 432.884,Z 255.45,A -85,B 0,C 180,E1 -9324.356,E2 -9324.356} C_VEL
LIN {X 0,Y 433.224,Z 248.359,A -85,B 0,C 180,E1 -9325.122,E2 -9325.122} C_VEL
LIN {X 0,Y 433.555,Z 239.986,A -85,B 0,C 180,E1 -9325.856,E2 -9325.856} C_VEL
LIN {X 0,Y 434.008,Z 230.106,A -85,B 0,C 180,E1 -9326.527,E2 -9326.527} C_VEL
LIN {X 0,Y 432.554,Z 220.435,A -85,B 0,C 180,E1 -9327.059,E2 -9327.059} C_VEL
LIN {X 0,Y 431.423,Z 214.694,A -85,B 0,C 180,E1 -9327.344,E2 -9327.344} C_VEL
LIN {X 0,Y 431.541,Z 209.661,A -85,B 0,C 180,E1 -9330.754,E2 -9330.754} C_VEL
LIN {X 0,Y 431.659,Z 205.07,A -85,B 0,C 180,E1 -9333.923,E2 -9333.923} C_VEL
LIN {X 0,Y 431.793,Z 200.657,A -85,B 0,C 180,E1 -9337.007,E2 -9337.007} C_VEL
LIN {X 0,Y 432.024,Z 195.56,A -85,B 0,C 180,E1 -9340.652,E2 -9340.652} C_VEL
LIN {X 0,Y 432.209,Z 191.008,A -85,B 0,C 180,E1 -9343.954,E2 -9343.954} C_VEL
LIN {X 0,Y 432.225,Z 188.414,A -85,B 0,C 180,E1 -9345.884,E2 -9345.884} C_VEL
LIN {X 0,Y 432.287,Z 187.458,A -85,B 0,C 180,E1 -9346.845,E2 -9346.845} C_VEL
LIN {X 0,Y 432.406,Z 187.439,A -85,B 0,C 180,E1 -9349.702,E2 -9349.702} C_VEL
LIN {X 0,Y 432.564,Z 187.422,A -85,B 0,C 180,E1 -9352.533,E2 -9352.533} C_VEL
LIN {X 0,Y 432.598,Z 187.418,A -85,B 0,C 180,E1 -9354.407,E2 -9354.407} C_VEL
LIN {X 0,Y 432.606,Z 187.414,A -85,B 0,C 180,E1 -9358.139,E2 -9358.139} C_VEL
LIN {X 0,Y 432.735,Z 187.396,A -85,B 0,C 180,E1 -9360.001,E2 -9360.001} C_VEL
LIN {X 0,Y 432.593,Z 187.412,A -85,B 0,C 180,E1 -9362.794,E2 -9362.794} C_VEL
LIN {X 0,Y 432.565,Z 187.417,A -85,B 0,C 180,E1 -9366.531,E2 -9366.531} C_VEL
LIN {X 0,Y 432.442,Z 187.434,A -85,B 0,C 180,E1 -9369.354,E2 -9369.354} C_VEL
LIN {X 0,Y 432.433,Z 187.434,A -85,B 0,C 180,E1 -9372.804,E2 -9372.804} C_VEL
LIN {X 0,Y 432.415,Z 187.436,A -85,B 0,C 180,E1 -9376.48,E2 -9376.48} C_VEL
LIN {X 0,Y 432.342,Z 187.445,A -85,B 0,C 180,E1 -9379.961,E2 -9379.961} C_VEL
LIN {X 0,Y 432.32,Z 187.449,A -85,B 0,C 180,E1 -9382.965,E2 -9382.965} C_VEL
LIN {X 0,Y 432.363,Z 187.441,A -85,B 0,C 180,E1 -9386.033,E2 -9386.033} C_VEL
LIN {X 0,Y 432.345,Z 187.444,A -85,B 0,C 180,E1 -9389.188,E2 -9389.188} C_VEL
LIN {X 0,Y 432.325,Z 187.447,A -85,B 0,C 180,E1 -9392.443,E2 -9392.443} C_VEL
LIN {X 0,Y 432.346,Z 187.445,A -85,B 0,C 180,E1 -9395.632,E2 -9395.632} C_VEL
LIN {X 0,Y 432.342,Z 187.444,A -85,B 0,C 180,E1 -9398.715,E2 -9398.715} C_VEL
LIN {X 0,Y 432.335,Z 187.448,A -85,B 0,C 180,E1 -9401.797,E2 -9401.797} C_VEL
LIN {X 0,Y 432.336,Z 187.448,A -85,B 0,C 180,E1 -9404.348,E2 -9404.348} C_VEL
LIN {X 0,Y 432.322,Z 187.45,A -85,B 0,C 180,E1 -9407.016,E2 -9407.016} C_VEL
LIN {X 0,Y 432.338,Z 187.446,A -85,B 0,C 180,E1 -9409.821,E2 -9409.821} C_VEL
LIN {X 0,Y 432.309,Z 187.454,A -85,B 0,C 180,E1 -9413.022,E2 -9413.022} C_VEL
LIN {X 0,Y 432.359,Z 187.458,A -85,B 0,C 180,E1 -9413.897,E2 -9413.897} C_VEL
LIN {X 0,Y 433.356,Z 192.77,A -85,B 0,C 180,E1 -9416.537,E2 -9416.537} C_VEL
LIN {X 0,Y 434.007,Z 197.596,A -85,B 0,C 180,E1 -9418.79,E2 -9418.79} C_VEL
LIN {X 0,Y 433.505,Z 204.046,A -85,B 0,C 180,E1 -9421.517,E2 -9421.517} C_VEL
LIN {X 0,Y 432.846,Z 212.715,A -85,B 0,C 180,E1 -9425.029,E2 -9425.029} C_VEL
LIN {X 0,Y 432.317,Z 221.791,A -85,B 0,C 180,E1 -9428.545,E2 -9428.545} C_VEL
LIN {X 0,Y 431.981,Z 229.613,A -85,B 0,C 180,E1 -9431.503,E2 -9431.503} C_VEL
LIN {X 0,Y 431.636,Z 238.871,A -85,B 0,C 180,E1 -9434.899,E2 -9434.899} C_VEL
LIN {X 0,Y 431.498,Z 244.29,A -85,B 0,C 180,E1 -9436.86,E2 -9436.86} C_VEL
LIN {X 0,Y 432.851,Z 255.212,A -85,B 0,C 180,E1 -9437.274,E2 -9437.274} C_VEL
LIN {X 0,Y 433.573,Z 265.796,A -85,B 0,C 180,E1 -9437.835,E2 -9437.835} C_VEL
LIN {X 0,Y 433.28,Z 274.585,A -85,B 0,C 180,E1 -9438.421,E2 -9438.421} C_VEL
LIN {X 0,Y 432.798,Z 282.975,A -85,B 0,C 180,E1 -9439.119,E2 -9439.119} C_VEL
LIN {X 0,Y 432.418,Z 290.92,A -85,B 0,C 180,E1 -9439.938,E2 -9439.938} C_VEL
LIN {X 0,Y 432.089,Z 298.353,A -85,B 0,C 180,E1 -9440.875,E2 -9440.875} C_VEL
LIN {X 0,Y 431.736,Z 305.898,A -85,B 0,C 180,E1 -9442.047,E2 -9442.047} C_VEL
LIN {X 0,Y 431.443,Z 312.793,A -85,B 0,C 180,E1 -9443.453,E2 -9443.453} C_VEL
LIN {X 0,Y 431.348,Z 318.03,A -85,B 0,C 180,E1 -9444.859,E2 -9444.859} C_VEL
LIN {X 0,Y 431.237,Z 321.875,A -85,B 0,C 180,E1 -9446.262,E2 -9446.262} C_VEL
LIN {X 0,Y 431.295,Z 323.64,A -85,B 0,C 180,E1 -9447.198,E2 -9447.198} C_VEL
LIN {X 0,Y 431.242,Z 324.892,A -85,B 0,C 180,E1 -9448.132,E2 -9448.132} C_VEL
LIN {X 0,Y 431.22,Z 325.659,A -85,B 0,C 180,E1 -9449.066,E2 -9449.066} C_VEL
LIN {X 0,Y 431.224,Z 325.947,A -85,B 0,C 180,E1 -9450,E2 -9450} C_VEL
LIN {X 0,Y 431.22,Z 325.651,A -85,B 0,C 180,E1 -9450.934,E2 -9450.934} C_VEL
LIN {X 0,Y 431.242,Z 324.823,A -85,B 0,C 180,E1 -9451.868,E2 -9451.868} C_VEL
LIN {X 0,Y 431.295,Z 323.508,A -85,B 0,C 180,E1 -9452.802,E2 -9452.802} C_VEL
LIN {X 0,Y 431.241,Z 320.518,A -85,B 0,C 180,E1 -9454.206,E2 -9454.206} C_VEL
LIN {X 0,Y 431.331,Z 316.234,A -85,B 0,C 180,E1 -9455.611,E2 -9455.611} C_VEL
LIN {X 0,Y 431.542,Z 310.264,A -85,B 0,C 180,E1 -9457.016,E2 -9457.016} C_VEL
LIN {X 0,Y 431.703,Z 305.302,A -85,B 0,C 180,E1 -9457.954,E2 -9457.954} C_VEL
LIN {X 0,Y 431.983,Z 299.315,A -85,B 0,C 180,E1 -9458.891,E2 -9458.891} C_VEL
LIN {X 0,Y 432.294,Z 292.02,A -85,B 0,C 180,E1 -9459.829,E2 -9459.829} C_VEL
LIN {X 0,Y 432.641,Z 284.218,A -85,B 0,C 180,E1 -9460.649,E2 -9460.649} C_VEL
LIN {X 0,Y 433.087,Z 276.006,A -85,B 0,C 180,E1 -9461.348,E2 -9461.348} C_VEL
LIN {X 0,Y 433.431,Z 265.574,A -85,B 0,C 180,E1 -9462.05,E2 -9462.05} C_VEL
LIN {X 0,Y 432.506,Z 254.277,A -85,B 0,C 180,E1 -9462.615,E2 -9462.615} C_VEL
LIN {X 0,Y 431.446,Z 244.763,A -85,B 0,C 180,E1 -9462.987,E2 -9462.987} C_VEL
LIN {X 0,Y 431.725,Z 236.015,A -85,B 0,C 180,E1 -9466.167,E2 -9466.167} C_VEL
LIN {X 0,Y 432.068,Z 227.319,A -85,B 0,C 180,E1 -9469.364,E2 -9469.364} C_VEL
LIN {X 0,Y 432.501,Z 217.744,A -85,B 0,C 180,E1 -9472.954,E2 -9472.954} C_VEL
LIN {X 0,Y 433.051,Z 208.781,A -85,B 0,C 180,E1 -9476.402,E2 -9476.402} C_VEL
LIN {X 0,Y 433.667,Z 200.607,A -85,B 0,C 180,E1 -9479.623,E2 -9479.623} C_VEL
LIN {X 0,Y 433.879,Z 196.675,A -85,B 0,C 180,E1 -9481.221,E2 -9481.221} C_VEL
LIN {X 0,Y 432.849,Z 190.034,A -85,B 0,C 180,E1 -9484.099,E2 -9484.099} C_VEL
LIN {X 0,Y 432.386,Z 187.44,A -85,B 0,C 180,E1 -9485.338,E2 -9485.338} C_VEL
LIN {X 0,Y 432.344,Z 187.445,A -85,B 0,C 180,E1 -9488.714,E2 -9488.714} C_VEL
LIN {X 0,Y 432.337,Z 187.444,A -85,B 0,C 180,E1 -9491.797,E2 -9491.797} C_VEL
LIN {X 0,Y 432.337,Z 187.447,A -85,B 0,C 180,E1 -9494.347,E2 -9494.347} C_VEL
LIN {X 0,Y 432.32,Z 187.445,A -85,B 0,C 180,E1 -9497.016,E2 -9497.016} C_VEL
LIN {X 0,Y 432.317,Z 187.448,A -85,B 0,C 180,E1 -9499.824,E2 -9499.824} C_VEL
LIN {X 0,Y 432.31,Z 187.447,A -85,B 0,C 180,E1 -9503.022,E2 -9503.022} C_VEL
LIN {X 0,Y 432.364,Z 187.443,A -85,B 0,C 180,E1 -9505.996,E2 -9505.996} C_VEL
LIN {X 0,Y 432.352,Z 187.442,A -85,B 0,C 180,E1 -9509.489,E2 -9509.489} C_VEL
LIN {X 0,Y 432.395,Z 187.436,A -85,B 0,C 180,E1 -9512.928,E2 -9512.928} C_VEL
LIN {X 0,Y 432.372,Z 187.442,A -85,B 0,C 180,E1 -9516.023,E2 -9516.023} C_VEL
LIN {X 0,Y 432.355,Z 187.442,A -85,B 0,C 180,E1 -9519.046,E2 -9519.046} C_VEL
LIN {X 0,Y 432.378,Z 187.441,A -85,B 0,C 180,E1 -9522.011,E2 -9522.011} C_VEL
LIN {X 0,Y 432.4,Z 187.436,A -85,B 0,C 180,E1 -9524.926,E2 -9524.926} C_VEL
LIN {X 0,Y 432.464,Z 187.429,A -85,B 0,C 180,E1 -9527.803,E2 -9527.803} C_VEL
LIN {X 0,Y 432.468,Z 187.429,A -85,B 0,C 180,E1 -9531.589,E2 -9531.589} C_VEL
LIN {X 0,Y 432.595,Z 187.41,A -85,B 0,C 180,E1 -9534.405,E2 -9534.405} C_VEL
LIN {X 0,Y 432.606,Z 187.409,A -85,B 0,C 180,E1 -9538.137,E2 -9538.137} C_VEL
LIN {X 0,Y 432.734,Z 187.395,A -85,B 0,C 180,E1 -9539.999,E2 -9539.999} C_VEL
LIN {X 0,Y 432.595,Z 187.414,A -85,B 0,C 180,E1 -9542.793,E2 -9542.793} C_VEL
LIN {X 0,Y 432.558,Z 187.417,A -85,B 0,C 180,E1 -9546.53,E2 -9546.53} C_VEL
LIN {X 0,Y 432.442,Z 187.431,A -85,B 0,C 180,E1 -9549.352,E2 -9549.352} C_VEL
LIN {X 0,Y 432.433,Z 187.434,A -85,B 0,C 180,E1 -9552.802,E2 -9552.802} C_VEL
LIN {X 0,Y 432.413,Z 187.436,A -85,B 0,C 180,E1 -9556.477,E2 -9556.477} C_VEL
LIN {X 0,Y 432.339,Z 187.444,A -85,B 0,C 180,E1 -9559.959,E2 -9559.959} C_VEL
LIN {X 0,Y 432.318,Z 187.448,A -85,B 0,C 180,E1 -9562.963,E2 -9562.963} C_VEL
LIN {X 0,Y 432.36,Z 187.443,A -85,B 0,C 180,E1 -9566.031,E2 -9566.031} C_VEL
LIN {X 0,Y 432.342,Z 187.443,A -85,B 0,C 180,E1 -9569.186,E2 -9569.186} C_VEL
LIN {X 0,Y 432.321,Z 187.448,A -85,B 0,C 180,E1 -9572.442,E2 -9572.442} C_VEL
LIN {X 0,Y 432.343,Z 187.443,A -85,B 0,C 180,E1 -9575.631,E2 -9575.631} C_VEL
LIN {X 0,Y 432.343,Z 187.443,A -85,B 0,C 180,E1 -9578.714,E2 -9578.714} C_VEL
LIN {X 0,Y 432.329,Z 187.446,A -85,B 0,C 180,E1 -9581.796,E2 -9581.796} C_VEL
LIN {X 0,Y 432.329,Z 187.446,A -85,B 0,C 180,E1 -9584.346,E2 -9584.346} C_VEL
LIN {X 0,Y 432.315,Z 187.445,A -85,B 0,C 180,E1 -9587.015,E2 -9587.015} C_VEL
LIN {X 0,Y 432.328,Z 187.448,A -85,B 0,C 180,E1 -9589.82,E2 -9589.82} C_VEL
LIN {X 0,Y 432.31,Z 187.447,A -85,B 0,C 180,E1 -9593.022,E2 -9593.022} C_VEL
LIN {X 0,Y 432.353,Z 187.444,A -85,B 0,C 180,E1 -9595.995,E2 -9595.995} C_VEL
LIN {X 0,Y 432.388,Z 187.439,A -85,B 0,C 180,E1 -9599.743,E2 -9599.743} C_VEL
LIN {X 0,Y 432.393,Z 187.439,A -85,B 0,C 180,E1 -9603.372,E2 -9603.372} C_VEL
LIN {X 0,Y 432.364,Z 187.441,A -85,B 0,C 180,E1 -9606.023,E2 -9606.023} C_VEL
LIN {X 0,Y 432.343,Z 187.445,A -85,B 0,C 180,E1 -9609.045,E2 -9609.045} C_VEL
LIN {X 0,Y 432.37,Z 187.439,A -85,B 0,C 180,E1 -9612.011,E2 -9612.011} C_VEL
LIN {X 0,Y 432.39,Z 187.439,A -85,B 0,C 180,E1 -9614.926,E2 -9614.926} C_VEL
LIN {X 0,Y 432.475,Z 187.427,A -85,B 0,C 180,E1 -9617.804,E2 -9617.804} C_VEL
LIN {X 0,Y 432.483,Z 187.427,A -85,B 0,C 180,E1 -9621.59,E2 -9621.59} C_VEL
LIN {X 0,Y 432.589,Z 187.413,A -85,B 0,C 180,E1 -9624.406,E2 -9624.406} C_VEL
LIN {X 0,Y 432.595,Z 187.411,A -85,B 0,C 180,E1 -9628.138,E2 -9628.138} C_VEL
LIN {X 0,Y 432.723,Z 187.396,A -85,B 0,C 180,E1 -9630,E2 -9630} C_VEL
LIN {X 0,Y 432.597,Z 187.413,A -85,B 0,C 180,E1 -9632.793,E2 -9632.793} C_VEL
LIN {X 0,Y 432.456,Z 187.429,A -85,B 0,C 180,E1 -9635.027,E2 -9635.027} C_VEL
LIN {X 0,Y 431.896,Z 187.499,A -85,B 0,C 180,E1 -9635.806,E2 -9635.806} C_VEL
LIN {X 0,Y 429.05,Z 187.854,A -85,B 0,C 180,E1 -9637.07,E2 -9637.07} C_VEL
LIN {X 0,Y 426.566,Z 188.164,A -85,B 0,C 180,E1 -9638.091,E2 -9638.091} C_VEL
LIN {X 0,Y 425.485,Z 188.298,A -85,B 0,C 180,E1 -9638.881,E2 -9638.881} C_VEL
LIN {X 0,Y 425.394,Z 188.308,A -85,B 0,C 180,E1 -9639.149,E2 -9639.149} C_VEL
LIN {X 0,Y 425.361,Z 188.316,A -85,B 0,C 180,E1 -9642.403,E2 -9642.403} C_VEL
LIN {X 0,Y 425.017,Z 188.417,A -85,B 0,C 180,E1 -9645.096,E2 -9645.096} C_VEL
LIN {X 0,Y 424.8,Z 192.957,A -85,B 0,C 180,E1 -9648.321,E2 -9648.321} C_VEL
LIN {X 0,Y 424.69,Z 197.289,A -85,B 0,C 180,E1 -9651.35,E2 -9651.35} C_VEL
LIN {X 0,Y 424.573,Z 201.794,A -85,B 0,C 180,E1 -9654.445,E2 -9654.445} C_VEL
LIN {X 0,Y 424.419,Z 206.477,A -85,B 0,C 180,E1 -9657.623,E2 -9657.623} C_VEL
LIN {X 0,Y 424.287,Z 211.39,A -85,B 0,C 180,E1 -9660.897,E2 -9660.897} C_VEL
LIN {X 0,Y 424.27,Z 214.36,A -85,B 0,C 180,E1 -9662.811,E2 -9662.811} C_VEL
LIN {X 0,Y 425.93,Z 224.351,A -85,B 0,C 180,E1 -9663.273,E2 -9663.273} C_VEL
LIN {X 0,Y 426.695,Z 230.587,A -85,B 0,C 180,E1 -9663.63,E2 -9663.63} C_VEL
LIN {X 0,Y 426.334,Z 239.902,A -85,B 0,C 180,E1 -9664.274,E2 -9664.274} C_VEL
LIN {X 0,Y 426.026,Z 247.589,A -85,B 0,C 180,E1 -9664.946,E2 -9664.946} C_VEL
LIN {X 0,Y 425.659,Z 255.604,A -85,B 0,C 180,E1 -9665.811,E2 -9665.811} C_VEL
LIN {X 0,Y 425.254,Z 263.017,A -85,B 0,C 180,E1 -9666.805,E2 -9666.805} C_VEL
LIN {X 0,Y 424.911,Z 270.072,A -85,B 0,C 180,E1 -9668.027,E2 -9668.027} C_VEL
LIN {X 0,Y 424.675,Z 274.461,A -85,B 0,C 180,E1 -9668.966,E2 -9668.966} C_VEL
LIN {X 0,Y 424.5,Z 278.069,A -85,B 0,C 180,E1 -9669.907,E2 -9669.907} C_VEL
LIN {X 0,Y 424.315,Z 281.137,A -85,B 0,C 180,E1 -9670.906,E2 -9670.906} C_VEL
LIN {X 0,Y 424.226,Z 283.297,A -85,B 0,C 180,E1 -9671.8,E2 -9671.8} C_VEL
LIN {X 0,Y 424.146,Z 285.517,A -85,B 0,C 180,E1 -9673.193,E2 -9673.193} C_VEL
LIN {X 0,Y 424.054,Z 286.568,A -85,B 0,C 180,E1 -9674.551,E2 -9674.551} C_VEL
LIN {X 0,Y 424.071,Z 286.55,A -85,B 0,C 180,E1 -9675.891,E2 -9675.891} C_VEL
LIN {X 0,Y 424.179,Z 285.502,A -85,B 0,C 180,E1 -9677.212,E2 -9677.212} C_VEL
LIN {X 0,Y 424.276,Z 283.438,A -85,B 0,C 180,E1 -9678.504,E2 -9678.504} C_VEL
LIN {X 0,Y 424.487,Z 280.246,A -85,B 0,C 180,E1 -9679.783,E2 -9679.783} C_VEL
LIN {X 0,Y 424.751,Z 275.904,A -85,B 0,C 180,E1 -9681.048,E2 -9681.048} C_VEL
LIN {X 0,Y 424.984,Z 271.886,A -85,B 0,C 180,E1 -9681.977,E2 -9681.977} C_VEL
LIN {X 0,Y 425.301,Z 266.374,A -85,B 0,C 180,E1 -9683.014,E2 -9683.014} C_VEL
LIN {X 0,Y 425.64,Z 259.888,A -85,B 0,C 180,E1 -9684.005,E2 -9684.005} C_VEL
LIN {X 0,Y 426.126,Z 251.358,A -85,B 0,C 180,E1 -9685.05,E2 -9685.05} C_VEL
LIN {X 0,Y 426.576,Z 241.853,A -85,B 0,C 180,E1 -9685.934,E2 -9685.934} C_VEL
LIN {X 0,Y 426.982,Z 233.575,A -85,B 0,C 180,E1 -9686.538,E2 -9686.538} C_VEL
LIN {X 0,Y 426.99,Z 229.132,A -85,B 0,C 180,E1 -9686.821,E2 -9686.821} C_VEL
LIN {X 0,Y 425.083,Z 218.791,A -85,B 0,C 180,E1 -9687.381,E2 -9687.381} C_VEL
LIN {X 0,Y 424.369,Z 215.005,A -85,B 0,C 180,E1 -9687.566,E2 -9687.566} C_VEL
LIN {X 0,Y 424.529,Z 209.547,A -85,B 0,C 180,E1 -9691.331,E2 -9691.331} C_VEL
LIN {X 0,Y 424.599,Z 205,A -85,B 0,C 180,E1 -9694.511,E2 -9694.511} C_VEL
LIN {X 0,Y 424.802,Z 200.275,A -85,B 0,C 180,E1 -9697.892,E2 -9697.892} C_VEL
LIN {X 0,Y 424.978,Z 196.393,A -85,B 0,C 180,E1 -9700.687,E2 -9700.687} C_VEL
LIN {X 0,Y 425.13,Z 192.357,A -85,B 0,C 180,E1 -9703.679,E2 -9703.679} C_VEL
LIN {X 0,Y 425.207,Z 188.466,A -85,B 0,C 180,E1 -9706.622,E2 -9706.622} C_VEL
LIN {X 0,Y 425.334,Z 188.322,A -85,B 0,C 180,E1 -9708.564,E2 -9708.564} C_VEL
LIN {X 0,Y 425.548,Z 188.296,A -85,B 0,C 180,E1 -9712.269,E2 -9712.269} C_VEL
LIN {X 0,Y 425.555,Z 188.296,A -85,B 0,C 180,E1 -9714.314,E2 -9714.314} C_VEL
LIN {X 0,Y 425.575,Z 188.29,A -85,B 0,C 180,E1 -9718.108,E2 -9718.108} C_VEL
LIN {X 0,Y 425.705,Z 188.272,A -85,B 0,C 180,E1 -9720.001,E2 -9720.001} C_VEL
LIN {X 0,Y 425.547,Z 188.29,A -85,B 0,C 180,E1 -9722.841,E2 -9722.841} C_VEL
LIN {X 0,Y 425.554,Z 188.291,A -85,B 0,C 180,E1 -9725.688,E2 -9725.688} C_VEL
LIN {X 0,Y 425.41,Z 188.308,A -85,B 0,C 180,E1 -9728.551,E2 -9728.551} C_VEL
LIN {X 0,Y 425.414,Z 188.308,A -85,B 0,C 180,E1 -9732.402,E2 -9732.402} C_VEL
LIN {X 0,Y 425.391,Z 188.312,A -85,B 0,C 180,E1 -9736.312,E2 -9736.312} C_VEL
LIN {X 0,Y 425.331,Z 188.319,A -85,B 0,C 180,E1 -9739.636,E2 -9739.636} C_VEL
LIN {X 0,Y 425.307,Z 188.321,A -85,B 0,C 180,E1 -9743.366,E2 -9743.366} C_VEL
LIN {X 0,Y 425.349,Z 188.316,A -85,B 0,C 180,E1 -9746.844,E2 -9746.844} C_VEL
LIN {X 0,Y 425.293,Z 188.323,A -85,B 0,C 180,E1 -9749.72,E2 -9749.72} C_VEL
LIN {X 0,Y 425.285,Z 188.323,A -85,B 0,C 180,E1 -9753.048,E2 -9753.048} C_VEL
LIN {X 0,Y 425.284,Z 188.324,A -85,B 0,C 180,E1 -9755.929,E2 -9755.929} C_VEL
LIN {X 0,Y 425.29,Z 188.325,A -85,B 0,C 180,E1 -9759.042,E2 -9759.042} C_VEL
LIN {X 0,Y 425.292,Z 188.325,A -85,B 0,C 180,E1 -9761.959,E2 -9761.959} C_VEL
LIN {X 0,Y 425.287,Z 188.326,A -85,B 0,C 180,E1 -9765.283,E2 -9765.283} C_VEL
LIN {X 0,Y 425.277,Z 188.327,A -85,B 0,C 180,E1 -9768.622,E2 -9768.622} C_VEL
LIN {X 0,Y 425.312,Z 188.321,A -85,B 0,C 180,E1 -9771.103,E2 -9771.103} C_VEL
LIN {X 0,Y 425.326,Z 188.514,A -85,B 0,C 180,E1 -9773.672,E2 -9773.672} C_VEL
LIN {X 0,Y 426.379,Z 194.017,A -85,B 0,C 180,E1 -9776.483,E2 -9776.483} C_VEL
LIN {X 0,Y 426.95,Z 197.656,A -85,B 0,C 180,E1 -9778.214,E2 -9778.214} C_VEL
LIN {X 0,Y 426.862,Z 201.33,A -85,B 0,C 180,E1 -9779.857,E2 -9779.857} C_VEL
LIN {X 0,Y 426.179,Z 208.614,A -85,B 0,C 180,E1 -9782.937,E2 -9782.937} C_VEL
LIN {X 0,Y 425.601,Z 216.47,A -85,B 0,C 180,E1 -9786.136,E2 -9786.136} C_VEL
LIN {X 0,Y 425.148,Z 224.233,A -85,B 0,C 180,E1 -9789.182,E2 -9789.182} C_VEL
LIN {X 0,Y 424.797,Z 232.062,A -85,B 0,C 180,E1 -9792.178,E2 -9792.178} C_VEL
LIN {X 0,Y 424.529,Z 239.984,A -85,B 0,C 180,E1 -9795.132,E2 -9795.132} C_VEL
LIN {X 0,Y 424.407,Z 244.01,A -85,B 0,C 180,E1 -9796.619,E2 -9796.619} C_VEL
LIN {X 0,Y 425.974,Z 256.626,A -85,B 0,C 180,E1 -9797.126,E2 -9797.126} C_VEL
LIN {X 0,Y 426.61,Z 265.742,A -85,B 0,C 180,E1 -9797.634,E2 -9797.634} C_VEL
LIN {X 0,Y 426.328,Z 274.466,A -85,B 0,C 180,E1 -9798.229,E2 -9798.229} C_VEL
LIN {X 0,Y 425.804,Z 282.809,A -85,B 0,C 180,E1 -9798.938,E2 -9798.938} C_VEL
LIN {X 0,Y 425.427,Z 290.72,A -85,B 0,C 180,E1 -9799.771,E2 -9799.771} C_VEL
LIN {X 0,Y 425.068,Z 298.125,A -85,B 0,C 180,E1 -9800.723,E2 -9800.723} C_VEL
LIN {X 0,Y 424.663,Z 305.645,A -85,B 0,C 180,E1 -9801.913,E2 -9801.913} C_VEL
LIN {X 0,Y 424.433,Z 311.549,A -85,B 0,C 180,E1 -9803.105,E2 -9803.105} C_VEL
LIN {X 0,Y 424.239,Z 316.2,A -85,B 0,C 180,E1 -9804.296,E2 -9804.296} C_VEL
LIN {X 0,Y 424.229,Z 319.226,A -85,B 0,C 180,E1 -9805.249,E2 -9805.249} C_VEL
LIN {X 0,Y 424.143,Z 321.583,A -85,B 0,C 180,E1 -9806.2,E2 -9806.2} C_VEL
LIN {X 0,Y 424.191,Z 323.338,A -85,B 0,C 180,E1 -9807.151,E2 -9807.151} C_VEL
LIN {X 0,Y 424.166,Z 324.58,A -85,B 0,C 180,E1 -9808.101,E2 -9808.101} C_VEL
LIN {X 0,Y 424.137,Z 325.337,A -85,B 0,C 180,E1 -9809.051,E2 -9809.051} C_VEL
LIN {X 0,Y 424.138,Z 325.617,A -85,B 0,C 180,E1 -9810,E2 -9810} C_VEL
LIN {X 0,Y 424.137,Z 325.319,A -85,B 0,C 180,E1 -9810.95,E2 -9810.95} C_VEL
LIN {X 0,Y 424.167,Z 324.48,A -85,B 0,C 180,E1 -9811.899,E2 -9811.899} C_VEL
LIN {X 0,Y 424.207,Z 323.152,A -85,B 0,C 180,E1 -9812.849,E2 -9812.849} C_VEL
LIN {X 0,Y 424.163,Z 320.148,A -85,B 0,C 180,E1 -9814.276,E2 -9814.276} C_VEL
LIN {X 0,Y 424.239,Z 315.841,A -85,B 0,C 180,E1 -9815.705,E2 -9815.705} C_VEL
LIN {X 0,Y 424.49,Z 309.838,A -85,B 0,C 180,E1 -9817.133,E2 -9817.133} C_VEL
LIN {X 0,Y 424.636,Z 304.849,A -85,B 0,C 180,E1 -9818.087,E2 -9818.087} C_VEL
LIN {X 0,Y 424.95,Z 298.833,A -85,B 0,C 180,E1 -9819.04,E2 -9819.04} C_VEL
LIN {X 0,Y 425.242,Z 291.498,A -85,B 0,C 180,E1 -9819.994,E2 -9819.994} C_VEL
LIN {X 0,Y 425.562,Z 284.882,A -85,B 0,C 180,E1 -9820.707,E2 -9820.707} C_VEL
LIN {X 0,Y 426.017,Z 276.877,A -85,B 0,C 180,E1 -9821.418,E2 -9821.418} C_VEL
LIN {X 0,Y 426.32,Z 268.595,A -85,B 0,C 180,E1 -9822.013,E2 -9822.013} C_VEL
LIN {X 0,Y 426.179,Z 262.536,A -85,B 0,C 180,E1 -9822.379,E2 -9822.379} C_VEL
LIN {X 0,Y 425.316,Z 252.581,A -85,B 0,C 180,E1 -9822.856,E2 -9822.856} C_VEL
LIN {X 0,Y 424.387,Z 244.63,A -85,B 0,C 180,E1 -9823.143,E2 -9823.143} C_VEL
LIN {X 0,Y 424.664,Z 235.992,A -85,B 0,C 180,E1 -9826.341,E2 -9826.341} C_VEL
LIN {X 0,Y 425.039,Z 226.641,A -85,B 0,C 180,E1 -9829.857,E2 -9829.857} C_VEL
LIN {X 0,Y 425.519,Z 217.522,A -85,B 0,C 180,E1 -9833.353,E2 -9833.353} C_VEL
LIN {X 0,Y 426.008,Z 209.599,A -85,B 0,C 180,E1 -9836.451,E2 -9836.451} C_VEL
LIN {X 0,Y 426.645,Z 201.735,A -85,B 0,C 180,E1 -9839.616,E2 -9839.616} C_VEL
LIN {X 0,Y 426.852,Z 198.116,A -85,B 0,C 180,E1 -9841.111,E2 -9841.111} C_VEL
LIN {X 0,Y 426.106,Z 192.548,A -85,B 0,C 180,E1 -9843.541,E2 -9843.541} C_VEL
LIN {X 0,Y 425.333,Z 188.319,A -85,B 0,C 180,E1 -9845.48,E2 -9845.48} C_VEL
LIN {X 0,Y 425.291,Z 188.326,A -85,B 0,C 180,E1 -9849.042,E2 -9849.042} C_VEL
LIN {X 0,Y 425.294,Z 188.322,A -85,B 0,C 180,E1 -9851.958,E2 -9851.958} C_VEL
LIN {X 0,Y 425.288,Z 188.322,A -85,B 0,C 180,E1 -9855.283,E2 -9855.283} C_VEL
LIN {X 0,Y 425.269,Z 188.326,A -85,B 0,C 180,E1 -9858.62,E2 -9858.62} C_VEL
LIN {X 0,Y 425.285,Z 188.32,A -85,B 0,C 180,E1 -9861.099,E2 -9861.099} C_VEL
LIN {X 0,Y 425.304,Z 188.32,A -85,B 0,C 180,E1 -9864.664,E2 -9864.664} C_VEL
LIN {X 0,Y 425.27,Z 188.327,A -85,B 0,C 180,E1 -9868.073,E2 -9868.073} C_VEL
LIN {X 0,Y 425.335,Z 188.317,A -85,B 0,C 180,E1 -9871.368,E2 -9871.368} C_VEL
LIN {X 0,Y 425.358,Z 188.315,A -85,B 0,C 180,E1 -9873.505,E2 -9873.505} C_VEL
LIN {X 0,Y 425.289,Z 188.321,A -85,B 0,C 180,E1 -9876.633,E2 -9876.633} C_VEL
LIN {X 0,Y 425.3,Z 188.323,A -85,B 0,C 180,E1 -9879.694,E2 -9879.694} C_VEL
LIN {X 0,Y 425.344,Z 188.314,A -85,B 0,C 180,E1 -9882.697,E2 -9882.697} C_VEL
LIN {X 0,Y 425.353,Z 188.316,A -85,B 0,C 180,E1 -9885.65,E2 -9885.65} C_VEL
LIN {X 0,Y 425.354,Z 188.313,A -85,B 0,C 180,E1 -9888.563,E2 -9888.563} C_VEL
LIN {X 0,Y 425.51,Z 188.294,A -85,B 0,C 180,E1 -9892.31,E2 -9892.31} C_VEL
LIN {X 0,Y 425.551,Z 188.288,A -85,B 0,C 180,E1 -9894.312,E2 -9894.312} C_VEL
LIN {X 0,Y 425.576,Z 188.284,A -85,B 0,C 180,E1 -9898.106,E2 -9898.106} C_VEL
LIN {X 0,Y 425.703,Z 188.27,A -85,B 0,C 180,E1 -9899.999,E2 -9899.999} C_VEL
LIN {X 0,Y 425.548,Z 188.292,A -85,B 0,C 180,E1 -9902.839,E2 -9902.839} C_VEL
LIN {X 0,Y 425.55,Z 188.288,A -85,B 0,C 180,E1 -9905.686,E2 -9905.686} C_VEL
LIN {X 0,Y 425.411,Z 188.308,A -85,B 0,C 180,E1 -9908.55,E2 -9908.55} C_VEL
LIN {X 0,Y 425.414,Z 188.307,A -85,B 0,C 180,E1 -9912.401,E2 -9912.401} C_VEL
LIN {X 0,Y 425.389,Z 188.31,A -85,B 0,C 180,E1 -9916.311,E2 -9916.311} C_VEL
LIN {X 0,Y 425.329,Z 188.316,A -85,B 0,C 180,E1 -9919.634,E2 -9919.634} C_VEL
LIN {X 0,Y 425.288,Z 188.324,A -85,B 0,C 180,E1 -9922.338,E2 -9922.338} C_VEL
LIN {X 0,Y 425.29,Z 188.321,A -85,B 0,C 180,E1 -9925.444,E2 -9925.444} C_VEL
LIN {X 0,Y 425.348,Z 188.313,A -85,B 0,C 180,E1 -9927.556,E2 -9927.556} C_VEL
LIN {X 0,Y 425.286,Z 188.323,A -85,B 0,C 180,E1 -9930.815,E2 -9930.815} C_VEL
LIN {X 0,Y 425.31,Z 188.321,A -85,B 0,C 180,E1 -9934.287,E2 -9934.287} C_VEL
LIN {X 0,Y 425.282,Z 188.324,A -85,B 0,C 180,E1 -9937.692,E2 -9937.692} C_VEL
LIN {X 0,Y 425.276,Z 188.325,A -85,B 0,C 180,E1 -9940.519,E2 -9940.519} C_VEL
LIN {X 0,Y 425.253,Z 188.325,A -85,B 0,C 180,E1 -9943.35,E2 -9943.35} C_VEL
LIN {X 0,Y 425.253,Z 188.325,A -85,B 0,C 180,E1 -9946.648,E2 -9946.648} C_VEL
LIN {X 0,Y 425.281,Z 188.326,A -85,B 0,C 180,E1 -9949.872,E2 -9949.872} C_VEL
LIN {X 0,Y 425.279,Z 188.323,A -85,B 0,C 180,E1 -9952.486,E2 -9952.486} C_VEL
LIN {X 0,Y 425.302,Z 188.322,A -85,B 0,C 180,E1 -9955.816,E2 -9955.816} C_VEL
LIN {X 0,Y 425.294,Z 188.324,A -85,B 0,C 180,E1 -9959.236,E2 -9959.236} C_VEL
LIN {X 0,Y 425.343,Z 188.314,A -85,B 0,C 180,E1 -9962.442,E2 -9962.442} C_VEL
LIN {X 0,Y 425.344,Z 188.317,A -85,B 0,C 180,E1 -9965.601,E2 -9965.601} C_VEL
LIN {X 0,Y 425.286,Z 188.322,A -85,B 0,C 180,E1 -9968.681,E2 -9968.681} C_VEL
LIN {X 0,Y 425.325,Z 188.318,A -85,B 0,C 180,E1 -9971.702,E2 -9971.702} C_VEL
LIN {X 0,Y 425.342,Z 188.317,A -85,B 0,C 180,E1 -9974.67,E2 -9974.67} C_VEL
LIN {X 0,Y 425.424,Z 188.306,A -85,B 0,C 180,E1 -9977.598,E2 -9977.598} C_VEL
LIN {X 0,Y 425.434,Z 188.305,A -85,B 0,C 180,E1 -9981.45,E2 -9981.45} C_VEL
LIN {X 0,Y 425.546,Z 188.289,A -85,B 0,C 180,E1 -9984.313,E2 -9984.313} C_VEL
LIN {X 0,Y 425.564,Z 188.287,A -85,B 0,C 180,E1 -9988.107,E2 -9988.107} C_VEL
LIN {X 0,Y 425.693,Z 188.271,A -85,B 0,C 180,E1 -9990,E2 -9990} C_VEL
LIN {X 0,Y 425.548,Z 188.291,A -85,B 0,C 180,E1 -9992.84,E2 -9992.84} C_VEL
LIN {X 0,Y 425.522,Z 188.294,A -85,B 0,C 180,E1 -9996.639,E2 -9996.639} C_VEL
LIN {X 0,Y 425.394,Z 188.308,A -85,B 0,C 180,E1 -9999.149,E2 -9999.149} C_VEL
LIN {X 0,Y 424.716,Z 188.395,A -85,B 0,C 180,E1 -9999.939,E2 -9999.939} C_VEL
LIN {X 0,Y 421.837,Z 188.751,A -85,B 0,C 180,E1 -10001.222,E2 -10001.222} C_VEL
LIN {X 0,Y 419.383,Z 189.06,A -85,B 0,C 180,E1 -10002.258,E2 -10002.258} C_VEL
LIN {X 0,Y 418.301,Z 189.192,A -85,B 0,C 180,E1 -10003.058,E2 -10003.058} C_VEL
LIN {X 0,Y 418.197,Z 189.204,A -85,B 0,C 180,E1 -10003.33,E2 -10003.33} C_VEL
LIN {X 0,Y 417.978,Z 189.255,A -85,B 0,C 180,E1 -10005.107,E2 -10005.107} C_VEL
LIN {X 0,Y 417.72,Z 194.177,A -85,B 0,C 180,E1 -10008.643,E2 -10008.643} C_VEL
LIN {X 0,Y 417.615,Z 198.563,A -85,B 0,C 180,E1 -10011.73,E2 -10011.73} C_VEL
LIN {X 0,Y 417.489,Z 203.112,A -85,B 0,C 180,E1 -10014.888,E2 -10014.888} C_VEL
LIN {X 0,Y 417.308,Z 207.885,A -85,B 0,C 180,E1 -10018.135,E2 -10018.135} C_VEL
LIN {X 0,Y 417.213,Z 212.831,A -85,B 0,C 180,E1 -10021.48,E2 -10021.48} C_VEL
LIN {X 0,Y 417.213,Z 214.56,A -85,B 0,C 180,E1 -10022.618,E2 -10022.618} C_VEL
LIN {X 0,Y 418.983,Z 225.39,A -85,B 0,C 180,E1 -10023.135,E2 -10023.135} C_VEL
LIN {X 0,Y 419.74,Z 230.915,A -85,B 0,C 180,E1 -10023.462,E2 -10023.462} C_VEL
LIN {X 0,Y 419.397,Z 238.856,A -85,B 0,C 180,E1 -10024.006,E2 -10024.006} C_VEL
LIN {X 0,Y 419.039,Z 247.572,A -85,B 0,C 180,E1 -10024.767,E2 -10024.767} C_VEL
LIN {X 0,Y 418.651,Z 255.978,A -85,B 0,C 180,E1 -10025.687,E2 -10025.687} C_VEL
LIN {X 0,Y 418.208,Z 263.509,A -85,B 0,C 180,E1 -10026.717,E2 -10026.717} C_VEL
LIN {X 0,Y 417.915,Z 269.639,A -85,B 0,C 180,E1 -10027.78,E2 -10027.78} C_VEL
LIN {X 0,Y 417.629,Z 274.736,A -85,B 0,C 180,E1 -10028.878,E2 -10028.878} C_VEL
LIN {X 0,Y 417.328,Z 279.672,A -85,B 0,C 180,E1 -10030.247,E2 -10030.247} C_VEL
LIN {X 0,Y 417.155,Z 283.279,A -85,B 0,C 180,E1 -10031.612,E2 -10031.612} C_VEL
LIN {X 0,Y 417.115,Z 284.67,A -85,B 0,C 180,E1 -10032.374,E2 -10032.374} C_VEL
LIN {X 0,Y 417.005,Z 286.384,A -85,B 0,C 180,E1 -10033.709,E2 -10033.709} C_VEL
LIN {X 0,Y 416.977,Z 287.074,A -85,B 0,C 180,E1 -10035.064,E2 -10035.064} C_VEL
LIN {X 0,Y 417.039,Z 286.64,A -85,B 0,C 180,E1 -10036.439,E2 -10036.439} C_VEL
LIN {X 0,Y 417.14,Z 285.019,A -85,B 0,C 180,E1 -10037.843,E2 -10037.843} C_VEL
LIN {X 0,Y 417.332,Z 282.18,A -85,B 0,C 180,E1 -10039.272,E2 -10039.272} C_VEL
LIN {X 0,Y 417.59,Z 277.938,A -85,B 0,C 180,E1 -10040.73,E2 -10040.73} C_VEL
LIN {X 0,Y 417.988,Z 271.785,A -85,B 0,C 180,E1 -10042.209,E2 -10042.209} C_VEL
LIN {X 0,Y 418.319,Z 266.06,A -85,B 0,C 180,E1 -10043.285,E2 -10043.285} C_VEL
LIN {X 0,Y 418.743,Z 259.214,A -85,B 0,C 180,E1 -10044.324,E2 -10044.324} C_VEL
LIN {X 0,Y 419.279,Z 250.096,A -85,B 0,C 180,E1 -10045.403,E2 -10045.403} C_VEL
LIN {X 0,Y 419.658,Z 241.92,A -85,B 0,C 180,E1 -10046.164,E2 -10046.164} C_VEL
LIN {X 0,Y 420.088,Z 233.682,A -85,B 0,C 180,E1 -10046.771,E2 -10046.771} C_VEL
LIN {X 0,Y 419.951,Z 229.423,A -85,B 0,C 180,E1 -10047.051,E2 -10047.051} C_VEL
LIN {X 0,Y 418.121,Z 219.522,A -85,B 0,C 180,E1 -10047.605,E2 -10047.605} C_VEL
LIN {X 0,Y 417.308,Z 215.295,A -85,B 0,C 180,E1 -10047.82,E2 -10047.82} C_VEL
LIN {X 0,Y 417.455,Z 210.608,A -85,B 0,C 180,E1 -10051.097,E2 -10051.097} C_VEL
LIN {X 0,Y 417.51,Z 206.439,A -85,B 0,C 180,E1 -10054.046,E2 -10054.046} C_VEL
LIN {X 0,Y 417.648,Z 203.475,A -85,B 0,C 180,E1 -10056.181,E2 -10056.181} C_VEL
LIN {X 0,Y 417.795,Z 199.167,A -85,B 0,C 180,E1 -10059.315,E2 -10059.315} C_VEL
LIN {X 0,Y 418.01,Z 195.063,A -85,B 0,C 180,E1 -10062.385,E2 -10062.385} C_VEL
LIN {X 0,Y 418.146,Z 191.088,A -85,B 0,C 180,E1 -10065.398,E2 -10065.398} C_VEL
LIN {X 0,Y 418.251,Z 189.207,A -85,B 0,C 180,E1 -10067.057,E2 -10067.057} C_VEL
LIN {X 0,Y 418.34,Z 189.189,A -85,B 0,C 180,E1 -10070.33,E2 -10070.33} C_VEL
LIN {X 0,Y 418.513,Z 189.172,A -85,B 0,C 180,E1 -10072.28,E2 -10072.28} C_VEL
LIN {X 0,Y 418.514,Z 189.173,A -85,B 0,C 180,E1 -10074.218,E2 -10074.218} C_VEL
LIN {X 0,Y 418.544,Z 189.166,A -85,B 0,C 180,E1 -10078.076,E2 -10078.076} C_VEL
LIN {X 0,Y 418.674,Z 189.148,A -85,B 0,C 180,E1 -10080.001,E2 -10080.001} C_VEL
LIN {X 0,Y 418.502,Z 189.167,A -85,B 0,C 180,E1 -10082.889,E2 -10082.889} C_VEL
LIN {X 0,Y 418.512,Z 189.169,A -85,B 0,C 180,E1 -10085.784,E2 -10085.784} C_VEL
LIN {X 0,Y 418.38,Z 189.183,A -85,B 0,C 180,E1 -10088.696,E2 -10088.696} C_VEL
LIN {X 0,Y 418.318,Z 189.192,A -85,B 0,C 180,E1 -10091.632,E2 -10091.632} C_VEL
LIN {X 0,Y 418.305,Z 189.192,A -85,B 0,C 180,E1 -10094.598,E2 -10094.598} C_VEL
LIN {X 0,Y 418.291,Z 189.195,A -85,B 0,C 180,E1 -10097.604,E2 -10097.604} C_VEL
LIN {X 0,Y 418.253,Z 189.2,A -85,B 0,C 180,E1 -10100.663,E2 -10100.663} C_VEL
LIN {X 0,Y 418.288,Z 189.195,A -85,B 0,C 180,E1 -10103.782,E2 -10103.782} C_VEL
LIN {X 0,Y 418.313,Z 189.192,A -85,B 0,C 180,E1 -10107.071,E2 -10107.071} C_VEL
LIN {X 0,Y 418.247,Z 189.201,A -85,B 0,C 180,E1 -10110.272,E2 -10110.272} C_VEL
LIN {X 0,Y 418.251,Z 189.199,A -85,B 0,C 180,E1 -10113.678,E2 -10113.678} C_VEL
LIN {X 0,Y 418.242,Z 189.201,A -85,B 0,C 180,E1 -10117.225,E2 -10117.225} C_VEL
LIN {X 0,Y 418.249,Z 189.201,A -85,B 0,C 180,E1 -10119.683,E2 -10119.683} C_VEL
LIN {X 0,Y 418.232,Z 189.205,A -85,B 0,C 180,E1 -10122.322,E2 -10122.322} C_VEL
LIN {X 0,Y 418.238,Z 189.205,A -85,B 0,C 180,E1 -10125.109,E2 -10125.109} C_VEL
LIN {X 0,Y 418.242,Z 189.203,A -85,B 0,C 180,E1 -10127.767,E2 -10127.767} C_VEL
LIN {X 0,Y 418.257,Z 189.201,A -85,B 0,C 180,E1 -10130.619,E2 -10130.619} C_VEL
LIN {X 0,Y 418.247,Z 189.334,A -85,B 0,C 180,E1 -10133.302,E2 -10133.302} C_VEL
LIN {X 0,Y 419.223,Z 194.178,A -85,B 0,C 180,E1 -10135.857,E2 -10135.857} C_VEL
LIN {X 0,Y 419.985,Z 198.843,A -85,B 0,C 180,E1 -10138.156,E2 -10138.156} C_VEL
LIN {X 0,Y 419.866,Z 202.573,A -85,B 0,C 180,E1 -10139.857,E2 -10139.857} C_VEL
LIN {X 0,Y 419.119,Z 210.048,A -85,B 0,C 180,E1 -10143.08,E2 -10143.08} C_VEL
LIN {X 0,Y 418.541,Z 217.672,A -85,B 0,C 180,E1 -10146.234,E2 -10146.234} C_VEL
LIN {X 0,Y 418.02,Z 226.685,A -85,B 0,C 180,E1 -10149.84,E2 -10149.84} C_VEL
LIN {X 0,Y 417.611,Z 235.831,A -85,B 0,C 180,E1 -10153.376,E2 -10153.376} C_VEL
LIN {X 0,Y 417.343,Z 243.715,A -85,B 0,C 180,E1 -10156.364,E2 -10156.364} C_VEL
LIN {X 0,Y 418.999,Z 256.661,A -85,B 0,C 180,E1 -10156.908,E2 -10156.908} C_VEL
LIN {X 0,Y 419.61,Z 265.695,A -85,B 0,C 180,E1 -10157.424,E2 -10157.424} C_VEL
LIN {X 0,Y 419.367,Z 274.364,A -85,B 0,C 180,E1 -10158.031,E2 -10158.031} C_VEL
LIN {X 0,Y 418.838,Z 282.668,A -85,B 0,C 180,E1 -10158.752,E2 -10158.752} C_VEL
LIN {X 0,Y 418.433,Z 290.548,A -85,B 0,C 180,E1 -10159.598,E2 -10159.598} C_VEL
LIN {X 0,Y 418.036,Z 297.93,A -85,B 0,C 180,E1 -10160.566,E2 -10160.566} C_VEL
LIN {X 0,Y 417.614,Z 305.425,A -85,B 0,C 180,E1 -10161.776,E2 -10161.776} C_VEL
LIN {X 0,Y 417.371,Z 311.295,A -85,B 0,C 180,E1 -10162.988,E2 -10162.988} C_VEL
LIN {X 0,Y 417.15,Z 315.927,A -85,B 0,C 180,E1 -10164.198,E2 -10164.198} C_VEL
LIN {X 0,Y 417.16,Z 318.943,A -85,B 0,C 180,E1 -10165.168,E2 -10165.168} C_VEL
LIN {X 0,Y 417.055,Z 321.296,A -85,B 0,C 180,E1 -10166.135,E2 -10166.135} C_VEL
LIN {X 0,Y 417.088,Z 323.038,A -85,B 0,C 180,E1 -10167.103,E2 -10167.103} C_VEL
LIN {X 0,Y 417.093,Z 324.271,A -85,B 0,C 180,E1 -10168.069,E2 -10168.069} C_VEL
LIN {X 0,Y 417.057,Z 325.016,A -85,B 0,C 180,E1 -10169.035,E2 -10169.035} C_VEL
LIN {X 0,Y 417.055,Z 325.286,A -85,B 0,C 180,E1 -10170,E2 -10170} C_VEL
LIN {X 0,Y 417.056,Z 324.988,A -85,B 0,C 180,E1 -10170.966,E2 -10170.966} C_VEL
LIN {X 0,Y 417.093,Z 324.136,A -85,B 0,C 180,E1 -10171.931,E2 -10171.931} C_VEL
LIN {X 0,Y 417.105,Z 322.792,A -85,B 0,C 180,E1 -10172.898,E2 -10172.898} C_VEL
LIN {X 0,Y 417.09,Z 319.774,A -85,B 0,C 180,E1 -10174.349,E2 -10174.349} C_VEL
LIN {X 0,Y 417.149,Z 315.441,A -85,B 0,C 180,E1 -10175.802,E2 -10175.802} C_VEL
LIN {X 0,Y 417.44,Z 309.404,A -85,B 0,C 180,E1 -10177.254,E2 -10177.254} C_VEL
LIN {X 0,Y 417.589,Z 304.389,A -85,B 0,C 180,E1 -10178.225,E2 -10178.225} C_VEL
LIN {X 0,Y 417.915,Z 298.343,A -85,B 0,C 180,E1 -10179.193,E2 -10179.193} C_VEL
LIN {X 0,Y 418.244,Z 290.971,A -85,B 0,C 180,E1 -10180.163,E2 -10180.163} C_VEL
LIN {X 0,Y 418.632,Z 283.077,A -85,B 0,C 180,E1 -10181.009,E2 -10181.009} C_VEL
LIN {X 0,Y 419.151,Z 273.247,A -85,B 0,C 180,E1 -10181.853,E2 -10181.853} C_VEL
LIN {X 0,Y 419.236,Z 264.04,A -85,B 0,C 180,E1 -10182.465,E2 -10182.465} C_VEL
LIN {X 0,Y 418.303,Z 252.853,A -85,B 0,C 180,E1 -10183.024,E2 -10183.024} C_VEL
LIN {X 0,Y 417.323,Z 244.348,A -85,B 0,C 180,E1 -10183.345,E2 -10183.345} C_VEL
LIN {X 0,Y 417.609,Z 235.688,A -85,B 0,C 180,E1 -10186.625,E2 -10186.625} C_VEL
LIN {X 0,Y 417.998,Z 226.489,A -85,B 0,C 180,E1 -10190.162,E2 -10190.162} C_VEL
LIN {X 0,Y 418.441,Z 218.573,A -85,B 0,C 180,E1 -10193.247,E2 -10193.247} C_VEL
LIN {X 0,Y 418.954,Z 210.699,A -85,B 0,C 180,E1 -10196.394,E2 -10196.394} C_VEL
LIN {X 0,Y 419.56,Z 203.312,A -85,B 0,C 180,E1 -10199.419,E2 -10199.419} C_VEL
LIN {X 0,Y 419.818,Z 198.638,A -85,B 0,C 180,E1 -10201.375,E2 -10201.375} C_VEL
LIN {X 0,Y 418.9,Z 192.514,A -85,B 0,C 180,E1 -10204.129,E2 -10204.129} C_VEL
LIN {X 0,Y 418.273,Z 189.197,A -85,B 0,C 180,E1 -10205.725,E2 -10205.725} C_VEL
LIN {X 0,Y 418.253,Z 189.202,A -85,B 0,C 180,E1 -10209.38,E2 -10209.38} C_VEL
LIN {X 0,Y 418.233,Z 189.202,A -85,B 0,C 180,E1 -10212.321,E2 -10212.321} C_VEL
LIN {X 0,Y 418.239,Z 189.2,A -85,B 0,C 180,E1 -10215.109,E2 -10215.109} C_VEL
LIN {X 0,Y 418.238,Z 189.2,A -85,B 0,C 180,E1 -10217.766,E2 -10217.766} C_VEL
LIN {X 0,Y 418.243,Z 189.198,A -85,B 0,C 180,E1 -10221.557,E2 -10221.557} C_VEL
LIN {X 0,Y 418.263,Z 189.195,A -85,B 0,C 180,E1 -10225.159,E2 -10225.159} C_VEL
LIN {X 0,Y 418.25,Z 189.199,A -85,B 0,C 180,E1 -10227.472,E2 -10227.472} C_VEL
LIN {X 0,Y 418.273,Z 189.195,A -85,B 0,C 180,E1 -10230.895,E2 -10230.895} C_VEL
LIN {X 0,Y 418.273,Z 189.198,A -85,B 0,C 180,E1 -10234.095,E2 -10234.095} C_VEL
LIN {X 0,Y 418.236,Z 189.201,A -85,B 0,C 180,E1 -10237.263,E2 -10237.263} C_VEL
LIN {X 0,Y 418.288,Z 189.194,A -85,B 0,C 180,E1 -10240.364,E2 -10240.364} C_VEL
LIN {X 0,Y 418.321,Z 189.191,A -85,B 0,C 180,E1 -10243.404,E2 -10243.404} C_VEL
LIN {X 0,Y 418.351,Z 189.186,A -85,B 0,C 180,E1 -10246.999,E2 -10246.999} C_VEL
LIN {X 0,Y 418.343,Z 189.186,A -85,B 0,C 180,E1 -10250.328,E2 -10250.328} C_VEL
LIN {X 0,Y 418.475,Z 189.172,A -85,B 0,C 180,E1 -10253.248,E2 -10253.248} C_VEL
LIN {X 0,Y 418.339,Z 189.19,A -85,B 0,C 180,E1 -10255.181,E2 -10255.181} C_VEL
LIN {X 0,Y 418.545,Z 189.16,A -85,B 0,C 180,E1 -10258.075,E2 -10258.075} C_VEL
LIN {X 0,Y 418.672,Z 189.146,A -85,B 0,C 180,E1 -10259.999,E2 -10259.999} C_VEL
LIN {X 0,Y 418.504,Z 189.17,A -85,B 0,C 180,E1 -10262.887,E2 -10262.887} C_VEL
LIN {X 0,Y 418.472,Z 189.172,A -85,B 0,C 180,E1 -10266.65,E2 -10266.65} C_VEL
LIN {X 0,Y 418.341,Z 189.186,A -85,B 0,C 180,E1 -10269.67,E2 -10269.67} C_VEL
LIN {X 0,Y 418.348,Z 189.189,A -85,B 0,C 180,E1 -10273,E2 -10273} C_VEL
LIN {X 0,Y 418.313,Z 189.194,A -85,B 0,C 180,E1 -10276.734,E2 -10276.734} C_VEL
LIN {X 0,Y 418.271,Z 189.195,A -85,B 0,C 180,E1 -10279.789,E2 -10279.789} C_VEL
LIN {X 0,Y 418.232,Z 189.203,A -85,B 0,C 180,E1 -10282.735,E2 -10282.735} C_VEL
LIN {X 0,Y 418.268,Z 189.197,A -85,B 0,C 180,E1 -10285.903,E2 -10285.903} C_VEL
LIN {X 0,Y 418.264,Z 189.197,A -85,B 0,C 180,E1 -10289.161,E2 -10289.161} C_VEL
LIN {X 0,Y 418.256,Z 189.199,A -85,B 0,C 180,E1 -10292.843,E2 -10292.843} C_VEL
LIN {X 0,Y 418.246,Z 189.201,A -85,B 0,C 180,E1 -10296.237,E2 -10296.237} C_VEL
LIN {X 0,Y 418.246,Z 189.199,A -85,B 0,C 180,E1 -10299.681,E2 -10299.681} C_VEL
LIN {X 0,Y 418.226,Z 189.203,A -85,B 0,C 180,E1 -10302.32,E2 -10302.32} C_VEL
LIN {X 0,Y 418.231,Z 189.201,A -85,B 0,C 180,E1 -10305.108,E2 -10305.108} C_VEL
LIN {X 0,Y 418.235,Z 189.203,A -85,B 0,C 180,E1 -10307.766,E2 -10307.766} C_VEL
LIN {X 0,Y 418.251,Z 189.201,A -85,B 0,C 180,E1 -10311.558,E2 -10311.558} C_VEL
LIN {X 0,Y 418.254,Z 189.199,A -85,B 0,C 180,E1 -10315.158,E2 -10315.158} C_VEL
LIN {X 0,Y 418.239,Z 189.202,A -85,B 0,C 180,E1 -10317.471,E2 -10317.471} C_VEL
LIN {X 0,Y 418.27,Z 189.196,A -85,B 0,C 180,E1 -10320.892,E2 -10320.892} C_VEL
LIN {X 0,Y 418.263,Z 189.197,A -85,B 0,C 180,E1 -10324.095,E2 -10324.095} C_VEL
LIN {X 0,Y 418.231,Z 189.203,A -85,B 0,C 180,E1 -10327.263,E2 -10327.263} C_VEL
LIN {X 0,Y 418.275,Z 189.195,A -85,B 0,C 180,E1 -10330.364,E2 -10330.364} C_VEL
LIN {X 0,Y 418.309,Z 189.193,A -85,B 0,C 180,E1 -10333.404,E2 -10333.404} C_VEL
LIN {X 0,Y 418.347,Z 189.189,A -85,B 0,C 180,E1 -10336.993,E2 -10336.993} C_VEL
LIN {X 0,Y 418.352,Z 189.185,A -85,B 0,C 180,E1 -10340.329,E2 -10340.329} C_VEL
LIN {X 0,Y 418.485,Z 189.171,A -85,B 0,C 180,E1 -10343.249,E2 -10343.249} C_VEL
LIN {X 0,Y 418.331,Z 189.19,A -85,B 0,C 180,E1 -10345.181,E2 -10345.181} C_VEL
LIN {X 0,Y 418.533,Z 189.162,A -85,B 0,C 180,E1 -10348.075,E2 -10348.075} C_VEL
LIN {X 0,Y 418.663,Z 189.147,A -85,B 0,C 180,E1 -10350,E2 -10350} C_VEL
LIN {X 0,Y 418.502,Z 189.169,A -85,B 0,C 180,E1 -10352.888,E2 -10352.888} C_VEL
LIN {X 0,Y 418.485,Z 189.171,A -85,B 0,C 180,E1 -10356.751,E2 -10356.751} C_VEL
LIN {X 0,Y 418.332,Z 189.188,A -85,B 0,C 180,E1 -10359.671,E2 -10359.671} C_VEL
LIN {X 0,Y 418.241,Z 189.2,A -85,B 0,C 180,E1 -10362.944,E2 -10362.944} C_VEL
LIN {X 0,Y 418.197,Z 189.204,A -85,B 0,C 180,E1 -10363.33,E2 -10363.33} C_VEL
LIN {X 0,Y 417.451,Z 189.437,A -85,B 0,C 180,E1 -10364.131,E2 -10364.131} C_VEL
LIN {X 0,Y 414.439,Z 190.58,A -85,B 0,C 180,E1 -10365.422,E2 -10365.422} C_VEL
LIN {X 0,Y 411.905,Z 191.928,A -85,B 0,C 180,E1 -10366.459,E2 -10366.459} C_VEL
LIN {X 0,Y 410.808,Z 193.051,A -85,B 0,C 180,E1 -10367.26,E2 -10367.26} C_VEL
LIN {X 0,Y 410.713,Z 193.427,A -85,B 0,C 180,E1 -10367.532,E2 -10367.532} C_VEL
LIN {X 0,Y 410.574,Z 198.336,A -85,B 0,C 180,E1 -10371.067,E2 -10371.067} C_VEL
LIN {X 0,Y 410.431,Z 203.707,A -85,B 0,C 180,E1 -10374.835,E2 -10374.835} C_VEL
LIN {X 0,Y 410.274,Z 207.62,A -85,B 0,C 180,E1 -10377.549,E2 -10377.549} C_VEL
LIN {X 0,Y 410.14,Z 212.764,A -85,B 0,C 180,E1 -10381.046,E2 -10381.046} C_VEL
LIN {X 0,Y 410.139,Z 214.923,A -85,B 0,C 180,E1 -10382.424,E2 -10382.424} C_VEL
LIN {X 0,Y 411.873,Z 225.325,A -85,B 0,C 180,E1 -10382.93,E2 -10382.93} C_VEL
LIN {X 0,Y 412.758,Z 231.472,A -85,B 0,C 180,E1 -10383.304,E2 -10383.304} C_VEL
LIN {X 0,Y 412.346,Z 240.884,A -85,B 0,C 180,E1 -10383.982,E2 -10383.982} C_VEL
LIN {X 0,Y 411.936,Z 249.817,A -85,B 0,C 180,E1 -10384.808,E2 -10384.808} C_VEL
LIN {X 0,Y 411.46,Z 259.376,A -85,B 0,C 180,E1 -10385.955,E2 -10385.955} C_VEL
LIN {X 0,Y 411.105,Z 264.741,A -85,B 0,C 180,E1 -10386.751,E2 -10386.751} C_VEL
LIN {X 0,Y 410.869,Z 270.044,A -85,B 0,C 180,E1 -10387.699,E2 -10387.699} C_VEL
LIN {X 0,Y 410.525,Z 275.803,A -85,B 0,C 180,E1 -10388.987,E2 -10388.987} C_VEL
LIN {X 0,Y 410.282,Z 279.621,A -85,B 0,C 180,E1 -10390.071,E2 -10390.071} C_VEL
LIN {X 0,Y 410.139,Z 282.381,A -85,B 0,C 180,E1 -10391.067,E2 -10391.067} C_VEL
LIN {X 0,Y 410.011,Z 285.279,A -85,B 0,C 180,E1 -10392.52,E2 -10392.52} C_VEL
LIN {X 0,Y 409.898,Z 286.936,A -85,B 0,C 180,E1 -10393.937,E2 -10393.937} C_VEL
LIN {X 0,Y 409.883,Z 287.396,A -85,B 0,C 180,E1 -10395.334,E2 -10395.334} C_VEL
LIN {X 0,Y 409.961,Z 286.76,A -85,B 0,C 180,E1 -10396.709,E2 -10396.709} C_VEL
LIN {X 0,Y 410.082,Z 285.118,A -85,B 0,C 180,E1 -10398.059,E2 -10398.059} C_VEL
LIN {X 0,Y 410.264,Z 282.469,A -85,B 0,C 180,E1 -10399.388,E2 -10399.388} C_VEL
LIN {X 0,Y 410.505,Z 278.769,A -85,B 0,C 180,E1 -10400.696,E2 -10400.696} C_VEL
LIN {X 0,Y 410.871,Z 273.833,A -85,B 0,C 180,E1 -10401.993,E2 -10401.993} C_VEL
LIN {X 0,Y 411.262,Z 267.442,A -85,B 0,C 180,E1 -10403.267,E2 -10403.267} C_VEL
LIN {X 0,Y 411.72,Z 260.47,A -85,B 0,C 180,E1 -10404.374,E2 -10404.374} C_VEL
LIN {X 0,Y 412.278,Z 251.589,A -85,B 0,C 180,E1 -10405.491,E2 -10405.491} C_VEL
LIN {X 0,Y 412.747,Z 242.829,A -85,B 0,C 180,E1 -10406.335,E2 -10406.335} C_VEL
LIN {X 0,Y 413.177,Z 235.103,A -85,B 0,C 180,E1 -10406.928,E2 -10406.928} C_VEL
LIN {X 0,Y 413.191,Z 231.499,A -85,B 0,C 180,E1 -10407.177,E2 -10407.177} C_VEL
LIN {X 0,Y 411.219,Z 220.5,A -85,B 0,C 180,E1 -10407.831,E2 -10407.831} C_VEL
LIN {X 0,Y 410.262,Z 215.597,A -85,B 0,C 180,E1 -10408.075,E2 -10408.075} C_VEL
LIN {X 0,Y 410.398,Z 210.97,A -85,B 0,C 180,E1 -10411.349,E2 -10411.349} C_VEL
LIN {X 0,Y 410.533,Z 205.731,A -85,B 0,C 180,E1 -10415.137,E2 -10415.137} C_VEL
LIN {X 0,Y 410.717,Z 201.978,A -85,B 0,C 180,E1 -10417.887,E2 -10417.887} C_VEL
LIN {X 0,Y 410.868,Z 197.785,A -85,B 0,C 180,E1 -10421.036,E2 -10421.036} C_VEL
LIN {X 0,Y 411.054,Z 193.773,A -85,B 0,C 180,E1 -10424.125,E2 -10424.125} C_VEL
LIN {X 0,Y 411.216,Z 190.084,A -85,B 0,C 180,E1 -10427.164,E2 -10427.164} C_VEL
LIN {X 0,Y 411.291,Z 190.068,A -85,B 0,C 180,E1 -10430.162,E2 -10430.162} C_VEL
LIN {X 0,Y 411.482,Z 190.048,A -85,B 0,C 180,E1 -10432.148,E2 -10432.148} C_VEL
LIN {X 0,Y 411.476,Z 190.05,A -85,B 0,C 180,E1 -10434.119,E2 -10434.119} C_VEL
LIN {X 0,Y 411.513,Z 190.042,A -85,B 0,C 180,E1 -10438.043,E2 -10438.043} C_VEL
LIN {X 0,Y 411.644,Z 190.023,A -85,B 0,C 180,E1 -10440.001,E2 -10440.001} C_VEL
LIN {X 0,Y 411.459,Z 190.044,A -85,B 0,C 180,E1 -10442.938,E2 -10442.938} C_VEL
LIN {X 0,Y 411.473,Z 190.046,A -85,B 0,C 180,E1 -10445.883,E2 -10445.883} C_VEL
LIN {X 0,Y 411.321,Z 190.062,A -85,B 0,C 180,E1 -10448.847,E2 -10448.847} C_VEL
LIN {X 0,Y 411.286,Z 190.068,A -85,B 0,C 180,E1 -10451.833,E2 -10451.833} C_VEL
LIN {X 0,Y 411.262,Z 190.07,A -85,B 0,C 180,E1 -10454.853,E2 -10454.853} C_VEL
LIN {X 0,Y 411.255,Z 190.071,A -85,B 0,C 180,E1 -10457.916,E2 -10457.916} C_VEL
LIN {X 0,Y 411.199,Z 190.079,A -85,B 0,C 180,E1 -10461.035,E2 -10461.035} C_VEL
LIN {X 0,Y 411.228,Z 190.076,A -85,B 0,C 180,E1 -10464.216,E2 -10464.216} C_VEL
LIN {X 0,Y 411.261,Z 190.071,A -85,B 0,C 180,E1 -10467.478,E2 -10467.478} C_VEL
LIN {X 0,Y 411.192,Z 190.079,A -85,B 0,C 180,E1 -10470.848,E2 -10470.848} C_VEL
LIN {X 0,Y 411.208,Z 190.077,A -85,B 0,C 180,E1 -10474.334,E2 -10474.334} C_VEL
LIN {X 0,Y 411.195,Z 190.08,A -85,B 0,C 180,E1 -10477.974,E2 -10477.974} C_VEL
LIN {X 0,Y 411.166,Z 190.085,A -85,B 0,C 180,E1 -10481.229,E2 -10481.229} C_VEL
